RoboDK station: kr30 cnc 070119 curve 7 axis test 2.rdk

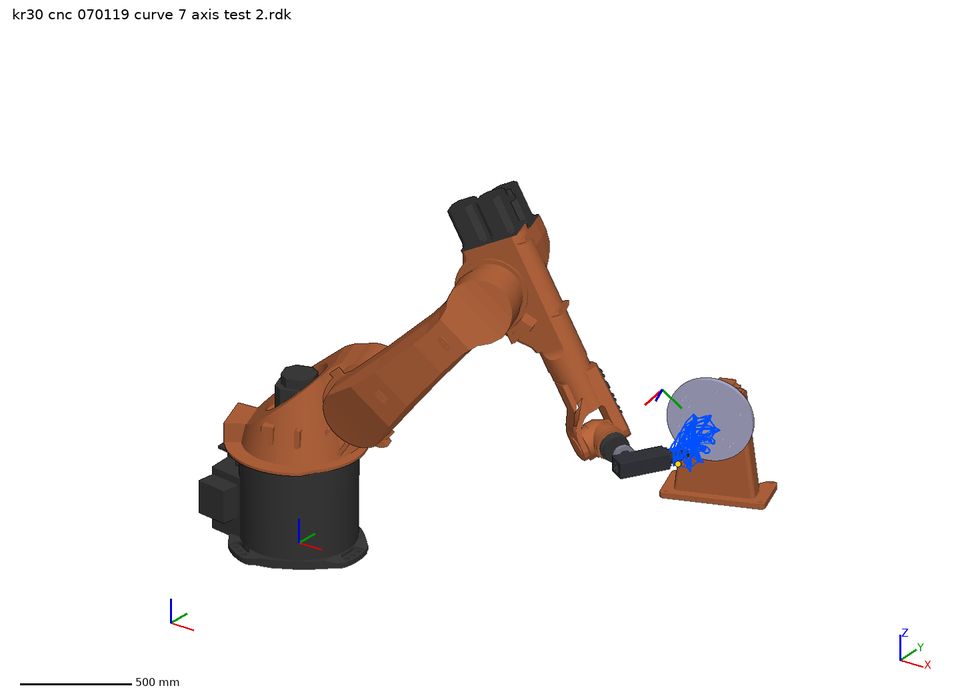
[picture v0: the station drawn from its stored meshes, robots at their saved joint values, targets as dots, program paths as lines]
Station kr30 cnc 070119 curve 7 axis test 2. Poses are relative to the parent item; angles as X-Y-Z fixed-axis rotations.
  - machining project Curve settings: C:/Temp/temp3/RhinoProject.stl | rotZ(0) | rotX(0)*rotY(0) | rotz(0) | onStart | onPathStart | onApproach | onPoint | onRetract | onFinish | onPathFinish | M_RunCode(%1)
  - frame KUKA KP1 MD250 Base at (0, 1000, 0) mm
    - robot KUKA KP1 MD250: 1 axes, payload 250 kg
        modified DH rows (alpha deg, a mm, theta deg, d mm): 0, 0, 0, 0
        base shift (1750, 1710, 820) mm, rotated rx 0 ry 90 rz -70 deg
        joint limits [-3600] to [3600]; home [0]; saved at [-1842.679]
      - frame Reference Rhino at (0, -260, 100) mm
        - object RhinoPart at (0, 0, 0) mm
  - frame KUKA KR 30 HA Base at (0, 2000, 0) mm
    - robot KUKA KR 30 HA: 6 axes, payload 30 kg, reach 2033 mm, repeatability 0.05 mm, weight 665 kg
        modified DH rows (alpha deg, a mm, theta deg, d mm): 0, 0, 0, 815; -90, 350, 0, 0; 0, 850, -90, 0; -90, 145, 0, 820; 90, 0, 0, 0; -90, 0, 180, 170
        joint limits [-185, -135, -120, -350, -119, -350] to [185, 35, 158, 350, 119, 350]; home [0, -90, 90, 0, 0, 0]; saved at [-17.768, -46.202, 111.125, 129.427, 73.448, 109.11]
      - tool 1/2" End Mill TCP, TCP at (337.71, -2.2, 160.57) mm, rotated rx 0 ry 90 rz 0 deg, size 415.8 x 102 x 153.6 mm
  - machining project RhinoPart Settings: rotZ(0) | rotX(0)*rotY(50) | rotz(0) | onStart | onPathStart | onApproach | onPoint | onRetract | onFinish | onPathFinish | M_RunCode(%1)
  - program RhinoPart (1340 instructions, listed below)
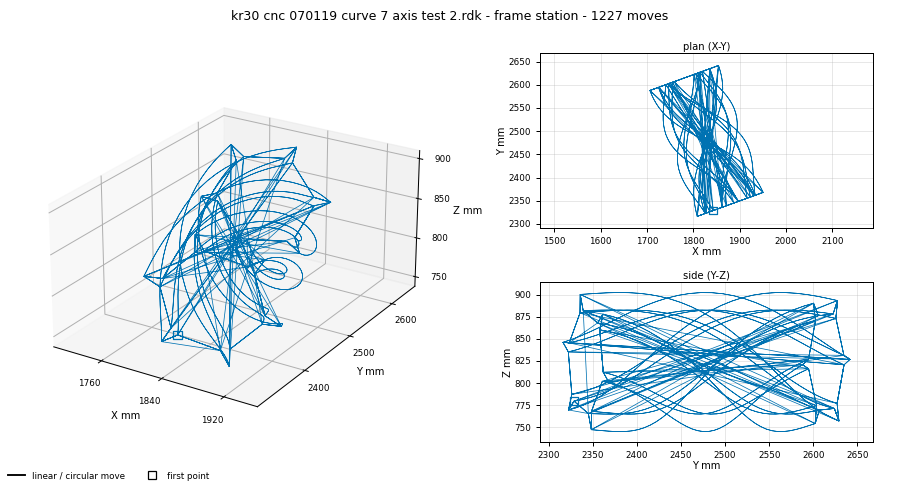
[picture p0: tool path of kr30 cnc 070119 curve 7 axis test 2.rdk in frame station, 1227 of 1227 moves have a stored position in this frame; points joined in program order, loops and branches not executed]

--- program RhinoPart (robot KUKA KR 30 HA) ---
  Set Ref.: Reference Rhino
  Set Tool: 1/2" End Mill TCP
  Show 1/2" End Mill TCP
  Set speed (1000.0 mm/s)
  MoveJ 1 to (58.93, 255.88, 290) mm, rotated rx 180 ry 50 rz -94 deg; joints [-8.613, -45.973, 108.773, 138.077, 69.074, 107.782, 4.002]
  MoveL 2 to (58.93, 255.88, 290) mm, rotated rx 180 ry 50 rz -94 deg; joints [-8.613, -45.973, 108.773, 138.077, 69.074, 107.782, 4.002]
  MoveL 3 to (58.93, 255.88, 290) mm, rotated rx 180 ry 50 rz -94 deg; joints [-8.613, -45.973, 108.773, 138.077, 69.074, 107.782, 4.002]
  Set speed (60.0 mm/s)
  MoveL 4 to (37.11, 300.24, 290) mm, rotated rx 180 ry 50 rz -42.69 deg; joints [-8.613, -46.208, 108.79, 138.021, 68.912, 107.938, -47.315]
  MoveL 5 to (-37.11, 208.63, 290) mm, rotated rx 180 ry 50 rz 144.16 deg; joints [-8.613, -45.739, 108.754, 138.132, 69.233, 107.629, 125.844]
  Set speed (60.0 mm/s)
  MoveL 6 to (-58.93, 252.99, 290) mm, rotated rx 180 ry 50 rz 96.78 deg; joints [-8.613, -45.958, 108.772, 138.081, 69.084, 107.773, 173.216]
  MoveL 7 to (21.11, 199.39, 290) mm, rotated rx 180 ry 50 rz -160.79 deg; joints [-8.613, -45.696, 108.75, 138.142, 69.263, 107.6, 70.794]
  Set speed (60.0 mm/s)
  MoveL 8 to (34.79, 183.72, 290) mm, rotated rx -180 ry 50 rz -155.49 deg; joints [-8.613, -44.618, 108.643, 138.382, 69.987, 106.912, 65.485]
  MoveL 9 to (21.11, 199.39, 290) mm, rotated rx -180 ry 50 rz -160.79 deg; joints [-8.613, -45.696, 108.75, 138.142, 69.263, 107.6, 70.794]
  Set speed (60.0 mm/s)
  MoveL 10 to (-28.22, 202.67, 290) mm, rotated rx 180 ry 50 rz 153.79 deg; joints [-8.613, -45.711, 108.751, 138.138, 69.253, 107.611, 116.207]
  MoveL 11 to (-43.85, 188.95, 290) mm, rotated rx -180 ry 50 rz 148.32 deg; joints [-8.613, -44.637, 108.645, 138.378, 69.974, 106.924, 121.679]
  Set speed (60.0 mm/s)
  MoveL 12 to (-28.22, 202.67, 290) mm, rotated rx -180 ry 50 rz 153.79 deg; joints [-8.613, -45.711, 108.751, 138.138, 69.253, 107.611, 116.207]
  MoveL 13 to (-43.85, 188.95, 290) mm, rotated rx -180 ry 50 rz 148.32 deg; joints [-8.613, -44.637, 108.645, 138.378, 69.974, 106.924, 121.679]
  Set speed (60.0 mm/s)
  MoveL 14 to (-37.11, 208.63, 290) mm, rotated rx 180 ry 50 rz 144.16 deg; joints [-8.613, -45.739, 108.754, 138.132, 69.233, 107.629, 125.844]
  MoveL 15 to (-78.63, 259.66, 290) mm, rotated rx -180 ry 50 rz 90.25 deg; joints [-8.613, -44.905, 108.674, 138.32, 69.797, 107.092, 179.755]
  Set speed (60.0 mm/s)
  MoveL 16 to (-58.93, 252.99, 290) mm, rotated rx 180 ry 50 rz 96.78 deg; joints [-8.613, -45.958, 108.772, 138.081, 69.084, 107.773, 173.216]
  MoveL 17 to (-78.63, 259.66, 290) mm, rotated rx 180 ry 50 rz 90.25 deg; joints [-8.613, -44.905, 108.674, 138.32, 69.797, 107.092, 179.755]
  Set speed (60.0 mm/s)
  MoveL 18 to (-58.22, 263.67, 290) mm, rotated rx -180 ry 50 rz 86.39 deg; joints [-8.613, -46.013, 108.776, 138.068, 69.046, 107.809, 183.606]
  MoveL 19 to (-30.72, 304.75, 290) mm, rotated rx -180 ry 50 rz 34.47 deg; joints [-8.613, -46.233, 108.792, 138.015, 68.894, 107.955, 235.533]
  Set speed (60.0 mm/s)
  MoveL 20 to (-58.22, 263.67, 290) mm, rotated rx -180 ry 50 rz 86.39 deg; joints [-8.613, -46.013, 108.776, 138.068, 69.046, 107.809, 183.606]
  MoveL 21 to (-30.72, 304.75, 290) mm, rotated rx -180 ry 50 rz 34.47 deg; joints [-8.613, -46.233, 108.792, 138.015, 68.894, 107.955, 235.533]
  Set speed (60.0 mm/s)
  MoveL 22 to (-34.79, 325.15, 290) mm, rotated rx 180 ry 50 rz 28.1 deg; joints [-8.613, -45.167, 108.701, 138.262, 69.621, 107.259, 241.899]
  MoveL 23 to (-21.11, 309.47, 290) mm, rotated rx 180 ry 50 rz 23.11 deg; joints [-8.613, -46.26, 108.794, 138.009, 68.876, 107.972, 246.89]
  Set speed (60.0 mm/s)
  MoveL 24 to (-34.79, 325.15, 290) mm, rotated rx 180 ry 50 rz 28.1 deg; joints [-8.613, -45.167, 108.701, 138.262, 69.621, 107.259, 241.899]
  MoveL 25 to (-21.11, 309.47, 290) mm, rotated rx 180 ry 50 rz 23.11 deg; joints [-8.613, -46.26, 108.794, 138.009, 68.876, 107.972, 246.89]
  Set speed (60.0 mm/s)
  MoveL 26 to (28.22, 306.19, 290) mm, rotated rx 180 ry 50 rz -31.42 deg; joints [-8.613, -46.241, 108.793, 138.013, 68.889, 107.96, 301.418]
  MoveL 27 to (43.85, 319.91, 290) mm, rotated rx 180 ry 50 rz -36.2 deg; joints [-8.613, -45.145, 108.699, 138.267, 69.635, 107.245, 306.197]
  Set speed (60.0 mm/s)
  MoveL 28 to (28.22, 306.19, 290) mm, rotated rx 180 ry 50 rz -31.42 deg; joints [-8.613, -46.241, 108.793, 138.013, 68.889, 107.96, 301.418]
  MoveL 29 to (43.85, 319.91, 290) mm, rotated rx 180 ry 50 rz -36.2 deg; joints [-8.613, -45.145, 108.699, 138.267, 69.635, 107.245, 306.197]
  Set speed (60.0 mm/s)
  MoveL 30 to (37.11, 300.24, 290) mm, rotated rx -180 ry 50 rz -42.69 deg; joints [-8.613, -46.208, 108.79, 138.021, 68.912, 107.938, 312.685]
  MoveL 31 to (78.63, 249.2, 290) mm, rotated rx -180 ry 50 rz -97.82 deg; joints [-8.613, -44.864, 108.67, 138.329, 69.824, 107.066, 367.819]
  Set speed (60.0 mm/s)
  MoveL 32 to (58.93, 255.88, 290) mm, rotated rx 180 ry 50 rz -94 deg; joints [-8.613, -45.973, 108.773, 138.077, 69.074, 107.782, 364.002]
  MoveL 33 to (78.63, 249.2, 290) mm, rotated rx 180 ry 50 rz -97.82 deg; joints [-8.613, -44.864, 108.67, 138.329, 69.824, 107.066, 367.819]
  Set speed (60.0 mm/s)
  MoveL 34 to (58.22, 245.2, 290) mm, rotated rx -180 ry 50 rz -104.27 deg; joints [-8.613, -45.919, 108.769, 138.09, 69.111, 107.747, 374.265]
  MoveL 35 to (30.72, 204.12, 290) mm, rotated rx -180 ry 50 rz -151.2 deg; joints [-8.613, -45.718, 108.752, 138.137, 69.248, 107.615, 421.204]
  Set speed (60.0 mm/s)
  MoveL 36 to (58.22, 245.2, 290) mm, rotated rx -180 ry 50 rz -104.27 deg; joints [-8.613, -45.919, 108.769, 138.09, 69.111, 107.747, 374.265]
  MoveL 37 to (30.72, 204.12, 290) mm, rotated rx -180 ry 50 rz -151.2 deg; joints [-8.613, -45.718, 108.752, 138.137, 69.248, 107.615, 421.204]
  Set speed (60.0 mm/s)
  MoveL 38 to (34.79, 183.72, 290) mm, rotated rx 180 ry 50 rz -155.49 deg; joints [-8.613, -44.618, 108.643, 138.382, 69.987, 106.912, 425.485]
  MoveL 39 to (-37.62, 299.82, 0) mm, rotated rx 180 ry 50 rz 43.38 deg; joints [-20.194, -47.371, 111.315, 126.82, 73.668, 110.587, 586.623]
  Set speed (60.0 mm/s)
  MoveL 40 to (10.16, 312.5, 0) mm, rotated rx 180 ry 50 rz -10.95 deg; joints [-20.194, -47.443, 111.32, 126.804, 73.628, 110.643, 640.953]
  MoveL 41 to (-37.62, 299.82, 0) mm, rotated rx 180 ry 50 rz 43.38 deg; joints [-20.194, -47.371, 111.315, 126.82, 73.668, 110.587, 586.623]
  Set speed (60.0 mm/s)
  MoveL 42 to (-55.59, 310.29, 0) mm, rotated rx 180 ry 50 rz 47.87 deg; joints [-20.194, -46.242, 111.219, 127.057, 74.288, 109.729, 582.13]
  MoveL 43 to (-45.21, 292.27, 0) mm, rotated rx -180 ry 50 rz 54.48 deg; joints [-20.194, -47.328, 111.312, 126.829, 73.692, 110.554, 575.516]
  Set speed (60.0 mm/s)
  MoveL 44 to (-55.59, 310.29, 0) mm, rotated rx 180 ry 50 rz 47.87 deg; joints [-20.194, -46.242, 111.219, 127.057, 74.288, 109.729, 582.13]
  MoveL 45 to (-45.21, 292.27, 0) mm, rotated rx -180 ry 50 rz 54.48 deg; joints [-20.194, -47.328, 111.312, 126.829, 73.692, 110.554, 575.516]
  Set speed (60.0 mm/s)
  MoveL 46 to (-58.12, 244.54, 0) mm, rotated rx -180 ry 50 rz 104.89 deg; joints [-20.194, -47.073, 111.293, 126.884, 73.834, 110.357, 525.106]
  MoveL 47 to (-76.17, 234.21, 0) mm, rotated rx 180 ry 50 rz 108.7 deg; joints [-20.194, -45.935, 111.187, 127.118, 74.455, 109.5, 521.297]
  Set speed (60.0 mm/s)
  MoveL 48 to (-58.12, 244.54, 0) mm, rotated rx 180 ry 50 rz 104.89 deg; joints [-20.194, -47.073, 111.293, 126.884, 73.834, 110.357, 525.106]
  MoveL 49 to (-76.17, 234.21, 0) mm, rotated rx 180 ry 50 rz 108.7 deg; joints [-20.194, -45.935, 111.187, 127.118, 74.455, 109.5, 521.297]
  Set speed (60.0 mm/s)
  MoveL 50 to (-55.37, 234.2, 0) mm, rotated rx 180 ry 50 rz 114.99 deg; joints [-20.194, -47.02, 111.288, 126.896, 73.863, 110.316, 515.014]
  MoveL 51 to (-20.49, 199.16, 0) mm, rotated rx -180 ry 50 rz 161.39 deg; joints [-20.194, -46.846, 111.274, 126.932, 73.959, 110.184, 468.615]
  Set speed (60.0 mm/s)
  MoveL 52 to (-55.37, 234.2, 0) mm, rotated rx 180 ry 50 rz 114.99 deg; joints [-20.194, -47.02, 111.288, 126.896, 73.863, 110.316, 515.014]
  MoveL 53 to (-20.49, 199.16, 0) mm, rotated rx -180 ry 50 rz 161.39 deg; joints [-20.194, -46.846, 111.274, 126.932, 73.959, 110.184, 468.615]
  Set speed (60.0 mm/s)
  MoveL 54 to (-20.57, 178.36, 0) mm, rotated rx -180 ry 50 rz 165.86 deg; joints [-20.194, -45.722, 111.164, 127.16, 74.569, 109.343, 464.144]
  MoveL 55 to (-10.16, 196.36, 0) mm, rotated rx -180 ry 50 rz 170.93 deg; joints [-20.194, -46.832, 111.273, 126.935, 73.966, 110.173, 459.071]
  Set speed (60.0 mm/s)
  MoveL 56 to (-20.57, 178.36, 0) mm, rotated rx -180 ry 50 rz 165.86 deg; joints [-20.194, -45.722, 111.164, 127.16, 74.569, 109.343, 464.144]
  MoveL 57 to (-10.16, 196.36, 0) mm, rotated rx -180 ry 50 rz 170.93 deg; joints [-20.194, -46.832, 111.273, 126.935, 73.966, 110.173, 459.071]
  Set speed (60.0 mm/s)
  MoveL 58 to (37.62, 209.05, 0) mm, rotated rx 180 ry 50 rz -143.56 deg; joints [-20.194, -46.894, 111.278, 126.922, 73.932, 110.22, 413.558]
  MoveL 59 to (55.59, 198.58, 0) mm, rotated rx 180 ry 50 rz -137.85 deg; joints [-20.194, -45.798, 111.172, 127.145, 74.528, 109.399, 407.85]
  Set speed (60.0 mm/s)
  MoveL 60 to (37.62, 209.05, 0) mm, rotated rx 180 ry 50 rz -143.56 deg; joints [-20.194, -46.894, 111.278, 126.922, 73.932, 110.22, 413.558]
  MoveL 61 to (55.59, 198.58, 0) mm, rotated rx 180 ry 50 rz -137.85 deg; joints [-20.194, -45.798, 111.172, 127.145, 74.528, 109.399, 407.85]
  Set speed (60.0 mm/s)
  MoveL 62 to (45.21, 216.6, 0) mm, rotated rx -180 ry 50 rz -133.83 deg; joints [-20.194, -46.931, 111.281, 126.914, 73.912, 110.249, 403.831]
  MoveL 63 to (58.12, 264.32, 0) mm, rotated rx -180 ry 50 rz -85.75 deg; joints [-20.194, -47.176, 111.301, 126.862, 73.776, 110.437, 355.746]
  Set speed (60.0 mm/s)
  MoveL 64 to (45.21, 216.6, 0) mm, rotated rx 180 ry 50 rz -133.83 deg; joints [-20.194, -46.931, 111.281, 126.914, 73.912, 110.249, 403.831]
  MoveL 65 to (58.12, 264.32, 0) mm, rotated rx -180 ry 50 rz -85.75 deg; joints [-20.194, -47.176, 111.301, 126.862, 73.776, 110.437, 355.746]
  Set speed (60.0 mm/s)
  MoveL 66 to (76.17, 274.65, 0) mm, rotated rx 180 ry 50 rz -79.11 deg; joints [-20.194, -46.096, 111.204, 127.086, 74.368, 109.619, 349.111]
  MoveL 67 to (55.37, 274.67, 0) mm, rotated rx 180 ry 50 rz -75.16 deg; joints [-20.194, -47.232, 111.305, 126.85, 73.745, 110.479, 345.162]
  Set speed (60.0 mm/s)
  MoveL 68 to (76.17, 274.65, 0) mm, rotated rx 180 ry 50 rz -79.11 deg; joints [-20.194, -46.096, 111.204, 127.086, 74.368, 109.619, 349.111]
  MoveL 69 to (55.37, 274.67, 0) mm, rotated rx 180 ry 50 rz -75.16 deg; joints [-20.194, -47.232, 111.305, 126.85, 73.745, 110.479, 345.162]
  Set speed (60.0 mm/s)
  MoveL 70 to (20.49, 309.71, 0) mm, rotated rx -180 ry 50 rz -22.4 deg; joints [-20.194, -47.427, 111.319, 126.808, 73.637, 110.631, 292.405]
  MoveL 71 to (20.57, 330.51, 0) mm, rotated rx -180 ry 50 rz -16.27 deg; joints [-20.194, -46.328, 111.227, 127.04, 74.242, 109.792, 286.267]
  Set speed (60.0 mm/s)
  MoveL 72 to (20.49, 309.71, 0) mm, rotated rx -180 ry 50 rz -22.4 deg; joints [-20.194, -47.427, 111.319, 126.808, 73.637, 110.631, 292.405]
  MoveL 73 to (20.57, 330.51, 0) mm, rotated rx -180 ry 50 rz -16.27 deg; joints [-20.194, -46.328, 111.227, 127.04, 74.242, 109.792, 286.267]
  Set speed (60.0 mm/s)
  MoveL 74 to (10.16, 312.5, 0) mm, rotated rx 180 ry 50 rz -10.95 deg; joints [-20.194, -47.443, 111.32, 126.804, 73.628, 110.643, 280.953]
  MoveL 75 to (-37.62, 299.82, 0) mm, rotated rx 180 ry 50 rz 43.38 deg; joints [-20.194, -47.371, 111.315, 126.82, 73.668, 110.587, 226.623]
  Set speed (60.0 mm/s)
  MoveL 76 to (-40.85, 296.93, 10) mm, rotated rx 180 ry 50 rz 47.89 deg; joints [-19.79, -47.354, 111.314, 127.219, 73.535, 110.463, 222.114]
  MoveL 77 to (-44.15, 293.5, 20) mm, rotated rx -180 ry 50 rz 52.81 deg; joints [-19.385, -47.332, 111.306, 127.618, 73.403, 110.338, 217.19]
  MoveL 78 to (-47.39, 289.5, 30) mm, rotated rx -180 ry 50 rz 58.1 deg; joints [-18.981, -47.304, 111.292, 128.017, 73.271, 110.213, 211.9]
  MoveL 79 to (-50.45, 284.92, 40) mm, rotated rx 180 ry 50 rz 63.71 deg; joints [-18.576, -47.27, 111.271, 128.417, 73.14, 110.088, 206.29]
  MoveL 80 to (-53.21, 279.8, 50) mm, rotated rx 180 ry 50 rz 69.59 deg; joints [-18.172, -47.231, 111.244, 128.817, 73.01, 109.962, 200.409]
  MoveL 81 to (-55.55, 274.16, 60) mm, rotated rx -180 ry 50 rz 75.7 deg; joints [-17.768, -47.186, 111.211, 129.217, 72.879, 109.836, 194.303]
  MoveL 82 to (-57.35, 268.08, 70) mm, rotated rx 180 ry 50 rz 81.99 deg; joints [-17.364, -47.136, 111.171, 129.617, 72.749, 109.711, 188.015]
  MoveL 83 to (-58.51, 261.62, 80) mm, rotated rx 180 ry 50 rz 88.41 deg; joints [-16.96, -47.082, 111.125, 130.017, 72.618, 109.586, 181.589]
  MoveL 84 to (-58.95, 254.91, 90) mm, rotated rx 180 ry 50 rz 94.94 deg; joints [-16.557, -47.024, 111.072, 130.417, 72.487, 109.462, 175.064]
  MoveL 85 to (-58.6, 248.05, 100) mm, rotated rx 180 ry 50 rz 101.52 deg; joints [-16.154, -46.962, 111.013, 130.816, 72.355, 109.339, 168.479]
  MoveL 86 to (-57.44, 241.19, 110) mm, rotated rx 180 ry 50 rz 108.13 deg; joints [-15.751, -46.899, 110.948, 131.215, 72.221, 109.219, 161.868]
  MoveL 87 to (-55.46, 234.45, 120) mm, rotated rx 180 ry 50 rz 114.74 deg; joints [-15.349, -46.833, 110.877, 131.613, 72.086, 109.101, 155.264]
  MoveL 88 to (-52.68, 227.97, 130) mm, rotated rx 180 ry 50 rz 121.3 deg; joints [-14.948, -46.766, 110.8, 132.009, 71.948, 108.986, 148.698]
  MoveL 89 to (-49.15, 221.88, 140) mm, rotated rx 180 ry 50 rz 127.8 deg; joints [-14.546, -46.699, 110.716, 132.405, 71.807, 108.874, 142.199]
  MoveL 90 to (-44.94, 216.28, 150) mm, rotated rx -180 ry 50 rz 134.21 deg; joints [-14.146, -46.632, 110.627, 132.799, 71.663, 108.766, 135.793]
  MoveL 91 to (-40.17, 211.29, 160) mm, rotated rx 180 ry 50 rz 140.49 deg; joints [-13.746, -46.565, 110.532, 133.191, 71.515, 108.662, 129.508]
  MoveL 92 to (-34.94, 206.95, 170) mm, rotated rx 180 ry 50 rz 146.63 deg; joints [-13.346, -46.498, 110.431, 133.582, 71.364, 108.561, 123.368]
  MoveL 93 to (-29.38, 203.32, 180) mm, rotated rx 180 ry 50 rz 152.6 deg; joints [-12.947, -46.432, 110.323, 133.971, 71.208, 108.465, 117.399]
  MoveL 94 to (-23.62, 200.42, 190) mm, rotated rx 180 ry 50 rz 158.37 deg; joints [-12.549, -46.367, 110.21, 134.359, 71.049, 108.372, 111.627]
  MoveL 95 to (-17.8, 198.23, 200) mm, rotated rx -180 ry 50 rz 163.92 deg; joints [-12.152, -46.303, 110.091, 134.744, 70.886, 108.283, 106.077]
  MoveL 96 to (-12.04, 196.73, 210) mm, rotated rx 180 ry 50 rz 169.22 deg; joints [-11.755, -46.239, 109.966, 135.128, 70.718, 108.198, 100.776]
  MoveL 97 to (-6.46, 195.84, 220) mm, rotated rx 180 ry 50 rz 174.25 deg; joints [-11.359, -46.175, 109.836, 135.51, 70.547, 108.115, 95.751]
  MoveL 98 to (-1.16, 195.49, 230) mm, rotated rx -180 ry 50 rz 178.97 deg; joints [-10.964, -46.111, 109.699, 135.891, 70.373, 108.036, 91.029]
  MoveL 99 to (3.78, 195.6, 240) mm, rotated rx -180 ry 50 rz -176.64 deg; joints [-10.57, -46.047, 109.556, 136.27, 70.195, 107.959, 86.641]
  MoveL 100 to (8.28, 196.07, 250) mm, rotated rx -180 ry 50 rz -172.62 deg; joints [-10.177, -45.981, 109.407, 136.647, 70.013, 107.885, 82.617]
  MoveL 101 to (12.3, 196.78, 260) mm, rotated rx 180 ry 50 rz -168.99 deg; joints [-9.784, -45.913, 109.252, 137.023, 69.829, 107.812, 78.987]
  MoveL 102 to (15.8, 197.64, 270) mm, rotated rx 180 ry 50 rz -165.79 deg; joints [-9.393, -45.843, 109.091, 137.397, 69.643, 107.74, 75.785]
  MoveL 103 to (18.74, 198.54, 280) mm, rotated rx 180 ry 50 rz -163.04 deg; joints [-9.003, -45.771, 108.924, 137.77, 69.454, 107.67, 73.043]
  MoveL 104 to (21.11, 199.39, 290) mm, rotated rx 180 ry 50 rz -160.79 deg; joints [-8.613, -45.696, 108.75, 138.142, 69.263, 107.6, 70.794]
  MoveL 105 to (10.16, 312.5, 0) mm, rotated rx 180 ry 50 rz -10.95 deg; joints [-20.194, -47.443, 111.32, 126.804, 73.628, 110.643, -79.047]
  Set speed (60.0 mm/s)
  MoveL 106 to (-37.62, 299.82, 0) mm, rotated rx 180 ry 50 rz 43.38 deg; joints [-20.194, -47.371, 111.315, 126.82, 73.668, 110.587, -133.377]
  MoveL 107 to (-28.22, 202.67, 290) mm, rotated rx -180 ry 50 rz 153.79 deg; joints [-8.613, -45.711, 108.751, 138.138, 69.253, 107.611, -243.793]
  Set speed (60.0 mm/s)
  MoveL 108 to (21.11, 199.39, 290) mm, rotated rx -180 ry 50 rz -160.79 deg; joints [-8.613, -45.696, 108.75, 138.142, 69.263, 107.6, -289.206]
  MoveL 109 to (-28.22, 202.67, 290) mm, rotated rx 180 ry 50 rz 153.79 deg; joints [-8.613, -45.711, 108.751, 138.138, 69.253, 107.611, -243.793]
  Set speed (60.0 mm/s)
  MoveL 110 to (-30.4, 203.93, 280) mm, rotated rx 180 ry 50 rz 151.53 deg; joints [-9.003, -45.797, 108.926, 137.764, 69.437, 107.687, -241.533]
  MoveL 111 to (-33, 205.58, 270) mm, rotated rx 180 ry 50 rz 148.77 deg; joints [-9.393, -45.881, 109.094, 137.388, 69.617, 107.765, -238.768]
  MoveL 112 to (-35.92, 207.69, 260) mm, rotated rx -180 ry 50 rz 145.53 deg; joints [-9.784, -45.965, 109.256, 137.011, 69.795, 107.846, -235.528]
  MoveL 113 to (-39.07, 210.28, 250) mm, rotated rx 180 ry 50 rz 141.84 deg; joints [-10.177, -46.049, 109.413, 136.631, 69.968, 107.93, -231.841]
  MoveL 114 to (-42.34, 213.41, 240) mm, rotated rx 180 ry 50 rz 137.73 deg; joints [-10.57, -46.132, 109.563, 136.25, 70.138, 108.017, -227.735]
  MoveL 115 to (-45.62, 217.1, 230) mm, rotated rx -180 ry 50 rz 133.24 deg; joints [-10.964, -46.215, 109.708, 135.867, 70.304, 108.106, -223.236]
  MoveL 116 to (-48.8, 221.36, 220) mm, rotated rx 180 ry 50 rz 128.37 deg; joints [-11.359, -46.299, 109.846, 135.482, 70.467, 108.199, -218.371]
  MoveL 117 to (-51.74, 226.19, 210) mm, rotated rx 180 ry 50 rz 123.16 deg; joints [-11.755, -46.382, 109.978, 135.096, 70.625, 108.296, -213.164]
  MoveL 118 to (-54.33, 231.55, 200) mm, rotated rx 180 ry 50 rz 117.64 deg; joints [-12.152, -46.466, 110.105, 134.707, 70.781, 108.395, -207.64]
  MoveL 119 to (-56.44, 237.4, 190) mm, rotated rx 180 ry 50 rz 111.82 deg; joints [-12.549, -46.549, 110.225, 134.318, 70.932, 108.498, -201.825]
  MoveL 120 to (-57.96, 243.66, 180) mm, rotated rx -180 ry 50 rz 105.74 deg; joints [-12.947, -46.632, 110.34, 133.926, 71.081, 108.604, -195.742]
  MoveL 121 to (-58.8, 250.25, 170) mm, rotated rx -180 ry 50 rz 99.42 deg; joints [-13.346, -46.715, 110.448, 133.533, 71.226, 108.713, -189.418]
  MoveL 122 to (-58.89, 257.04, 160) mm, rotated rx 180 ry 50 rz 92.88 deg; joints [-13.746, -46.795, 110.55, 133.139, 71.37, 108.825, -182.877]
  MoveL 123 to (-58.18, 263.92, 150) mm, rotated rx 180 ry 50 rz 86.15 deg; joints [-14.146, -46.874, 110.646, 132.744, 71.511, 108.939, -176.149]
  MoveL 124 to (-56.65, 270.74, 140) mm, rotated rx 180 ry 50 rz 79.26 deg; joints [-14.546, -46.951, 110.736, 132.348, 71.65, 109.055, -169.263]
  MoveL 125 to (-54.3, 277.38, 130) mm, rotated rx 180 ry 50 rz 72.25 deg; joints [-14.948, -47.023, 110.82, 131.951, 71.789, 109.171, -162.251]
  MoveL 126 to (-51.17, 283.7, 120) mm, rotated rx 180 ry 50 rz 65.15 deg; joints [-15.349, -47.092, 110.897, 131.554, 71.927, 109.289, -155.149]
  MoveL 127 to (-47.33, 289.58, 110) mm, rotated rx -180 ry 50 rz 57.99 deg; joints [-15.751, -47.156, 110.968, 131.157, 72.065, 109.407, -147.994]
  MoveL 128 to (-42.85, 294.92, 100) mm, rotated rx 180 ry 50 rz 50.83 deg; joints [-16.154, -47.214, 111.032, 130.76, 72.203, 109.524, -140.828]
  MoveL 129 to (-37.86, 299.62, 90) mm, rotated rx -180 ry 50 rz 43.7 deg; joints [-16.557, -47.266, 111.09, 130.363, 72.342, 109.641, -133.695]
  MoveL 130 to (-32.46, 303.64, 80) mm, rotated rx -180 ry 50 rz 36.64 deg; joints [-16.96, -47.312, 111.141, 129.966, 72.482, 109.757, -126.643]
  MoveL 131 to (-26.8, 306.94, 70) mm, rotated rx -180 ry 50 rz 29.72 deg; joints [-17.364, -47.351, 111.186, 129.569, 72.622, 109.871, -119.72]
  MoveL 132 to (-21, 309.52, 60) mm, rotated rx 180 ry 50 rz 22.98 deg; joints [-17.768, -47.383, 111.225, 129.173, 72.764, 109.984, -112.977]
  MoveL 133 to (-15.19, 311.39, 50) mm, rotated rx -180 ry 50 rz 16.46 deg; joints [-18.172, -47.408, 111.257, 128.777, 72.907, 110.096, -106.464]
  MoveL 134 to (-9.5, 312.61, 40) mm, rotated rx 180 ry 50 rz 10.23 deg; joints [-18.576, -47.426, 111.282, 128.382, 73.05, 110.207, -100.231]
  MoveL 135 to (-4.03, 313.25, 30) mm, rotated rx -180 ry 50 rz 4.33 deg; joints [-18.981, -47.439, 111.301, 127.987, 73.194, 110.316, -94.327]
  MoveL 136 to (1.12, 313.37, 20) mm, rotated rx 180 ry 50 rz -1.2 deg; joints [-19.385, -47.445, 111.314, 127.593, 73.339, 110.425, -88.799]
  MoveL 137 to (5.87, 313.09, 10) mm, rotated rx -180 ry 50 rz -6.31 deg; joints [-19.79, -47.446, 111.32, 127.198, 73.484, 110.534, -83.692]
  MoveL 138 to (10.16, 312.5, 0) mm, rotated rx 180 ry 50 rz -10.95 deg; joints [-20.194, -47.443, 111.32, 126.804, 73.628, 110.643, -79.047]
  MoveL 139 to (-37.62, 299.82, 0) mm, rotated rx 180 ry 50 rz 43.38 deg; joints [-20.194, -47.371, 111.315, 126.82, 73.668, 110.587, -133.377]
  Set speed (60.0 mm/s)
  MoveL 140 to (-40.85, 296.93, 10) mm, rotated rx 180 ry 50 rz 47.89 deg; joints [-19.79, -47.354, 111.314, 127.219, 73.535, 110.463, -137.886]
  MoveL 141 to (-44.15, 293.5, 20) mm, rotated rx -180 ry 50 rz 52.81 deg; joints [-19.385, -47.332, 111.306, 127.618, 73.403, 110.338, -142.81]
  MoveL 142 to (-47.39, 289.5, 30) mm, rotated rx -180 ry 50 rz 58.1 deg; joints [-18.981, -47.304, 111.292, 128.017, 73.271, 110.213, -148.1]
  MoveL 143 to (-50.45, 284.92, 40) mm, rotated rx 180 ry 50 rz 63.71 deg; joints [-18.576, -47.27, 111.271, 128.417, 73.14, 110.088, -153.71]
  MoveL 144 to (-53.21, 279.8, 50) mm, rotated rx 180 ry 50 rz 69.59 deg; joints [-18.172, -47.231, 111.244, 128.817, 73.01, 109.962, -159.591]
  MoveL 145 to (-55.55, 274.16, 60) mm, rotated rx -180 ry 50 rz 75.7 deg; joints [-17.768, -47.186, 111.211, 129.217, 72.879, 109.836, -165.697]
  MoveL 146 to (-57.35, 268.08, 70) mm, rotated rx 180 ry 50 rz 81.99 deg; joints [-17.364, -47.136, 111.171, 129.617, 72.749, 109.711, -171.985]
  MoveL 147 to (-58.51, 261.62, 80) mm, rotated rx -180 ry 50 rz 88.41 deg; joints [-16.96, -47.082, 111.125, 130.017, 72.618, 109.586, -178.411]
  MoveL 148 to (-58.95, 254.91, 90) mm, rotated rx 180 ry 50 rz 94.94 deg; joints [-16.557, -47.024, 111.072, 130.417, 72.487, 109.462, -184.936]
  MoveL 149 to (-58.6, 248.05, 100) mm, rotated rx 180 ry 50 rz 101.52 deg; joints [-16.154, -46.962, 111.013, 130.816, 72.355, 109.339, -191.521]
  MoveL 150 to (-57.44, 241.19, 110) mm, rotated rx 180 ry 50 rz 108.13 deg; joints [-15.751, -46.899, 110.948, 131.215, 72.221, 109.219, -198.132]
  MoveL 151 to (-55.46, 234.45, 120) mm, rotated rx 180 ry 50 rz 114.74 deg; joints [-15.349, -46.833, 110.877, 131.613, 72.086, 109.101, -204.736]
  MoveL 152 to (-52.68, 227.97, 130) mm, rotated rx 180 ry 50 rz 121.3 deg; joints [-14.948, -46.766, 110.8, 132.009, 71.948, 108.986, -211.302]
  MoveL 153 to (-49.15, 221.88, 140) mm, rotated rx 180 ry 50 rz 127.8 deg; joints [-14.546, -46.699, 110.716, 132.405, 71.807, 108.874, -217.801]
  MoveL 154 to (-44.94, 216.28, 150) mm, rotated rx 180 ry 50 rz 134.21 deg; joints [-14.146, -46.632, 110.627, 132.799, 71.663, 108.766, -224.207]
  MoveL 155 to (-40.17, 211.29, 160) mm, rotated rx 180 ry 50 rz 140.49 deg; joints [-13.746, -46.565, 110.532, 133.191, 71.515, 108.662, -230.492]
  MoveL 156 to (-34.94, 206.95, 170) mm, rotated rx 180 ry 50 rz 146.63 deg; joints [-13.346, -46.498, 110.431, 133.582, 71.364, 108.561, -236.632]
  MoveL 157 to (-29.38, 203.32, 180) mm, rotated rx 180 ry 50 rz 152.6 deg; joints [-12.947, -46.432, 110.323, 133.971, 71.208, 108.465, -242.601]
  MoveL 158 to (-23.62, 200.42, 190) mm, rotated rx -180 ry 50 rz 158.37 deg; joints [-12.549, -46.367, 110.21, 134.359, 71.049, 108.372, -248.373]
  MoveL 159 to (-17.8, 198.23, 200) mm, rotated rx -180 ry 50 rz 163.92 deg; joints [-12.152, -46.303, 110.091, 134.744, 70.886, 108.283, -253.923]
  MoveL 160 to (-12.04, 196.73, 210) mm, rotated rx 180 ry 50 rz 169.22 deg; joints [-11.755, -46.239, 109.966, 135.128, 70.718, 108.198, -259.224]
  MoveL 161 to (-6.46, 195.84, 220) mm, rotated rx -180 ry 50 rz 174.25 deg; joints [-11.359, -46.175, 109.836, 135.51, 70.547, 108.115, -264.249]
  MoveL 162 to (-1.16, 195.49, 230) mm, rotated rx 180 ry 50 rz 178.97 deg; joints [-10.964, -46.111, 109.699, 135.891, 70.373, 108.036, -268.971]
  MoveL 163 to (3.78, 195.6, 240) mm, rotated rx 180 ry 50 rz -176.64 deg; joints [-10.57, -46.047, 109.556, 136.27, 70.195, 107.959, -273.359]
  MoveL 164 to (8.28, 196.07, 250) mm, rotated rx 180 ry 50 rz -172.62 deg; joints [-10.177, -45.981, 109.407, 136.647, 70.013, 107.885, -277.383]
  MoveL 165 to (12.3, 196.78, 260) mm, rotated rx 180 ry 50 rz -168.99 deg; joints [-9.784, -45.913, 109.252, 137.023, 69.829, 107.812, -281.013]
  MoveL 166 to (15.8, 197.64, 270) mm, rotated rx 180 ry 50 rz -165.79 deg; joints [-9.393, -45.843, 109.091, 137.397, 69.643, 107.74, -284.215]
  MoveL 167 to (18.74, 198.54, 280) mm, rotated rx 180 ry 50 rz -163.04 deg; joints [-9.003, -45.771, 108.924, 137.77, 69.454, 107.67, -286.957]
  MoveL 168 to (21.11, 199.39, 290) mm, rotated rx 180 ry 50 rz -160.79 deg; joints [-8.613, -45.696, 108.75, 138.142, 69.263, 107.6, -289.206]
  MoveL 169 to (34.79, 183.72, 290) mm, rotated rx -180 ry 50 rz -155.49 deg; joints [-8.613, -44.618, 108.643, 138.382, 69.987, 106.912, -294.515]
  Set speed (60.0 mm/s)
  MoveL 170 to (21.11, 199.39, 290) mm, rotated rx -180 ry 50 rz -160.79 deg; joints [-8.613, -45.696, 108.75, 138.142, 69.263, 107.6, -289.206]
  MoveL 171 to (-55.59, 310.29, 0) mm, rotated rx -180 ry 50 rz 47.87 deg; joints [-20.194, -46.242, 111.219, 127.057, 74.288, 109.729, -137.87]
  Set speed (60.0 mm/s)
  MoveL 172 to (-37.62, 299.82, 0) mm, rotated rx 180 ry 50 rz 43.38 deg; joints [-20.194, -47.371, 111.315, 126.82, 73.668, 110.587, -133.377]
  MoveL 173 to (34.79, 183.72, 290) mm, rotated rx -180 ry 50 rz -155.49 deg; joints [-8.613, -44.618, 108.643, 138.382, 69.987, 106.912, -294.515]
  Set speed (60.0 mm/s)
  MoveL 174 to (31.73, 182.3, 280) mm, rotated rx 180 ry 50 rz -157.79 deg; joints [-9.003, -44.69, 108.816, 138.01, 70.176, 106.975, -292.214]
  MoveL 175 to (27.92, 180.74, 270) mm, rotated rx 180 ry 50 rz -160.59 deg; joints [-9.393, -44.76, 108.983, 137.637, 70.362, 107.039, -289.407]
  MoveL 176 to (23.38, 179.17, 260) mm, rotated rx 180 ry 50 rz -163.87 deg; joints [-9.784, -44.826, 109.144, 137.263, 70.547, 107.104, -286.13]
  MoveL 177 to (18.11, 177.74, 250) mm, rotated rx -180 ry 50 rz -167.58 deg; joints [-10.177, -44.89, 109.298, 136.887, 70.729, 107.171, -282.417]
  MoveL 178 to (12.17, 176.57, 240) mm, rotated rx 180 ry 50 rz -171.7 deg; joints [-10.57, -44.952, 109.447, 136.51, 70.908, 107.239, -278.3]
  MoveL 179 to (5.61, 175.83, 230) mm, rotated rx -180 ry 50 rz -176.19 deg; joints [-10.964, -45.013, 109.589, 136.131, 71.084, 107.309, -273.813]
  MoveL 180 to (-1.49, 175.64, 220) mm, rotated rx -180 ry 50 rz 178.99 deg; joints [-11.359, -45.073, 109.726, 135.751, 71.257, 107.381, -268.987]
  MoveL 181 to (-9.03, 176.15, 210) mm, rotated rx -180 ry 50 rz 173.85 deg; joints [-11.755, -45.133, 109.856, 135.369, 71.426, 107.456, -263.854]
  MoveL 182 to (-16.88, 177.46, 200) mm, rotated rx 180 ry 50 rz 168.44 deg; joints [-12.152, -45.193, 109.981, 134.985, 71.591, 107.535, -258.444]
  MoveL 183 to (-24.89, 179.66, 190) mm, rotated rx 180 ry 50 rz 162.78 deg; joints [-12.549, -45.254, 110.1, 134.6, 71.752, 107.617, -252.785]
  MoveL 184 to (-32.91, 182.83, 180) mm, rotated rx -180 ry 50 rz 156.91 deg; joints [-12.947, -45.316, 110.213, 134.212, 71.909, 107.702, -246.906]
  MoveL 185 to (-40.75, 186.98, 170) mm, rotated rx -180 ry 50 rz 150.84 deg; joints [-13.346, -45.378, 110.321, 133.823, 72.062, 107.792, -240.836]
  MoveL 186 to (-48.24, 192.12, 160) mm, rotated rx 180 ry 50 rz 144.6 deg; joints [-13.746, -45.442, 110.422, 133.433, 72.21, 107.886, -234.602]
  MoveL 187 to (-55.2, 198.19, 150) mm, rotated rx -180 ry 50 rz 138.23 deg; joints [-14.146, -45.506, 110.518, 133.04, 72.355, 107.983, -228.231]
  MoveL 188 to (-61.48, 205.13, 140) mm, rotated rx -180 ry 50 rz 131.75 deg; joints [-14.546, -45.571, 110.608, 132.647, 72.496, 108.085, -221.752]
  MoveL 189 to (-66.92, 212.81, 130) mm, rotated rx 180 ry 50 rz 125.19 deg; joints [-14.948, -45.636, 110.692, 132.251, 72.634, 108.19, -215.192]
  MoveL 190 to (-71.41, 221.1, 120) mm, rotated rx -180 ry 50 rz 118.58 deg; joints [-15.349, -45.701, 110.77, 131.855, 72.768, 108.299, -208.581]
  MoveL 191 to (-74.87, 229.83, 110) mm, rotated rx 180 ry 50 rz 111.95 deg; joints [-15.751, -45.765, 110.842, 131.457, 72.9, 108.41, -201.949]
  MoveL 192 to (-77.24, 238.83, 100) mm, rotated rx 180 ry 50 rz 105.33 deg; joints [-16.154, -45.828, 110.908, 131.058, 73.03, 108.525, -195.327]
  MoveL 193 to (-78.53, 247.91, 90) mm, rotated rx -180 ry 50 rz 98.75 deg; joints [-16.557, -45.889, 110.968, 130.659, 73.157, 108.642, -188.75]
  MoveL 194 to (-78.77, 256.9, 80) mm, rotated rx -180 ry 50 rz 92.25 deg; joints [-16.96, -45.947, 111.022, 130.259, 73.284, 108.76, -182.251]
  MoveL 195 to (-78, 265.63, 70) mm, rotated rx -180 ry 50 rz 85.87 deg; joints [-17.364, -46.001, 111.069, 129.859, 73.41, 108.88, -175.868]
  MoveL 196 to (-76.35, 273.96, 60) mm, rotated rx 180 ry 50 rz 79.64 deg; joints [-17.768, -46.051, 111.11, 129.458, 73.535, 109.001, -169.641]
  MoveL 197 to (-73.92, 281.75, 50) mm, rotated rx -180 ry 50 rz 73.61 deg; joints [-18.172, -46.097, 111.144, 129.057, 73.66, 109.122, -163.608]
  MoveL 198 to (-70.87, 288.9, 40) mm, rotated rx -180 ry 50 rz 67.81 deg; joints [-18.576, -46.137, 111.172, 128.657, 73.785, 109.244, -157.812]
  MoveL 199 to (-67.34, 295.36, 30) mm, rotated rx 180 ry 50 rz 62.3 deg; joints [-18.981, -46.172, 111.194, 128.256, 73.91, 109.365, -152.296]
  MoveL 200 to (-63.51, 301.08, 20) mm, rotated rx 180 ry 50 rz 57.1 deg; joints [-19.385, -46.201, 111.208, 127.856, 74.036, 109.487, -147.105]
  MoveL 201 to (-59.54, 306.05, 10) mm, rotated rx 180 ry 50 rz 52.28 deg; joints [-19.79, -46.225, 111.217, 127.456, 74.162, 109.608, -142.281]
  MoveL 202 to (-55.59, 310.29, 0) mm, rotated rx 180 ry 50 rz 47.87 deg; joints [-20.194, -46.242, 111.219, 127.057, 74.288, 109.729, -137.87]
  MoveL 203 to (34.79, 183.72, 290) mm, rotated rx -180 ry 50 rz -155.49 deg; joints [-8.613, -44.618, 108.643, 138.382, 69.987, 106.912, -294.515]
  Set speed (60.0 mm/s)
  MoveL 204 to (30.72, 204.12, 290) mm, rotated rx -180 ry 50 rz -151.2 deg; joints [-8.613, -45.718, 108.752, 138.137, 69.248, 107.615, -298.796]
  MoveL 205 to (-55.59, 310.29, 0) mm, rotated rx -180 ry 50 rz 47.87 deg; joints [-20.194, -46.242, 111.219, 127.057, 74.288, 109.729, -137.87]
  Set speed (60.0 mm/s)
  MoveL 206 to (-45.21, 292.27, 0) mm, rotated rx -180 ry 50 rz 54.48 deg; joints [-20.194, -47.328, 111.312, 126.829, 73.692, 110.554, -144.484]
  MoveL 207 to (-55.59, 310.29, 0) mm, rotated rx -180 ry 50 rz 47.87 deg; joints [-20.194, -46.242, 111.219, 127.057, 74.288, 109.729, -137.87]
  Set speed (60.0 mm/s)
  MoveL 208 to (-59.54, 306.05, 10) mm, rotated rx 180 ry 50 rz 52.28 deg; joints [-19.79, -46.225, 111.217, 127.456, 74.162, 109.608, -142.281]
  MoveL 209 to (-63.51, 301.08, 20) mm, rotated rx -180 ry 50 rz 57.1 deg; joints [-19.385, -46.201, 111.208, 127.856, 74.036, 109.487, -147.105]
  MoveL 210 to (-67.34, 295.36, 30) mm, rotated rx 180 ry 50 rz 62.3 deg; joints [-18.981, -46.172, 111.194, 128.256, 73.91, 109.365, -152.296]
  MoveL 211 to (-70.87, 288.9, 40) mm, rotated rx 180 ry 50 rz 67.81 deg; joints [-18.576, -46.137, 111.172, 128.657, 73.785, 109.244, -157.812]
  MoveL 212 to (-73.92, 281.75, 50) mm, rotated rx -180 ry 50 rz 73.61 deg; joints [-18.172, -46.097, 111.144, 129.057, 73.66, 109.122, -163.608]
  MoveL 213 to (-76.35, 273.96, 60) mm, rotated rx -180 ry 50 rz 79.64 deg; joints [-17.768, -46.051, 111.11, 129.458, 73.535, 109.001, -169.641]
  MoveL 214 to (-78, 265.63, 70) mm, rotated rx -180 ry 50 rz 85.87 deg; joints [-17.364, -46.001, 111.069, 129.859, 73.41, 108.88, -175.868]
  MoveL 215 to (-78.77, 256.9, 80) mm, rotated rx 180 ry 50 rz 92.25 deg; joints [-16.96, -45.947, 111.022, 130.259, 73.284, 108.76, -182.251]
  MoveL 216 to (-78.53, 247.91, 90) mm, rotated rx 180 ry 50 rz 98.75 deg; joints [-16.557, -45.889, 110.968, 130.659, 73.157, 108.642, -188.75]
  MoveL 217 to (-77.24, 238.83, 100) mm, rotated rx 180 ry 50 rz 105.33 deg; joints [-16.154, -45.828, 110.908, 131.058, 73.03, 108.525, -195.327]
  MoveL 218 to (-74.87, 229.83, 110) mm, rotated rx 180 ry 50 rz 111.95 deg; joints [-15.751, -45.765, 110.842, 131.457, 72.9, 108.41, -201.949]
  MoveL 219 to (-71.41, 221.1, 120) mm, rotated rx -180 ry 50 rz 118.58 deg; joints [-15.349, -45.701, 110.77, 131.855, 72.768, 108.299, -208.581]
  MoveL 220 to (-66.92, 212.81, 130) mm, rotated rx -180 ry 50 rz 125.19 deg; joints [-14.948, -45.636, 110.692, 132.251, 72.634, 108.19, -215.192]
  MoveL 221 to (-61.48, 205.13, 140) mm, rotated rx 180 ry 50 rz 131.75 deg; joints [-14.546, -45.571, 110.608, 132.647, 72.496, 108.085, -221.752]
  MoveL 222 to (-55.2, 198.19, 150) mm, rotated rx -180 ry 50 rz 138.23 deg; joints [-14.146, -45.506, 110.518, 133.04, 72.355, 107.983, -228.231]
  MoveL 223 to (-48.24, 192.12, 160) mm, rotated rx 180 ry 50 rz 144.6 deg; joints [-13.746, -45.442, 110.422, 133.433, 72.21, 107.886, -234.602]
  MoveL 224 to (-40.75, 186.98, 170) mm, rotated rx 180 ry 50 rz 150.84 deg; joints [-13.346, -45.378, 110.321, 133.823, 72.062, 107.792, -240.836]
  MoveL 225 to (-32.91, 182.83, 180) mm, rotated rx 180 ry 50 rz 156.91 deg; joints [-12.947, -45.316, 110.213, 134.212, 71.909, 107.702, -246.906]
  MoveL 226 to (-24.89, 179.66, 190) mm, rotated rx -180 ry 50 rz 162.78 deg; joints [-12.549, -45.254, 110.1, 134.6, 71.752, 107.617, -252.785]
  MoveL 227 to (-16.88, 177.46, 200) mm, rotated rx -180 ry 50 rz 168.44 deg; joints [-12.152, -45.193, 109.981, 134.985, 71.591, 107.535, -258.444]
  MoveL 228 to (-9.03, 176.15, 210) mm, rotated rx -180 ry 50 rz 173.85 deg; joints [-11.755, -45.133, 109.856, 135.369, 71.426, 107.456, -263.854]
  MoveL 229 to (-1.49, 175.64, 220) mm, rotated rx -180 ry 50 rz 178.99 deg; joints [-11.359, -45.073, 109.726, 135.751, 71.257, 107.381, -268.987]
  MoveL 230 to (5.61, 175.83, 230) mm, rotated rx -180 ry 50 rz -176.19 deg; joints [-10.964, -45.013, 109.589, 136.131, 71.084, 107.309, -273.813]
  MoveL 231 to (12.17, 176.57, 240) mm, rotated rx 180 ry 50 rz -171.7 deg; joints [-10.57, -44.952, 109.447, 136.51, 70.908, 107.239, -278.3]
  MoveL 232 to (18.11, 177.74, 250) mm, rotated rx -180 ry 50 rz -167.58 deg; joints [-10.177, -44.89, 109.298, 136.887, 70.729, 107.171, -282.417]
  MoveL 233 to (23.38, 179.17, 260) mm, rotated rx -180 ry 50 rz -163.87 deg; joints [-9.784, -44.826, 109.144, 137.263, 70.547, 107.104, -286.13]
  MoveL 234 to (27.92, 180.74, 270) mm, rotated rx 180 ry 50 rz -160.59 deg; joints [-9.393, -44.76, 108.983, 137.637, 70.362, 107.039, -289.407]
  MoveL 235 to (31.73, 182.3, 280) mm, rotated rx 180 ry 50 rz -157.79 deg; joints [-9.003, -44.69, 108.816, 138.01, 70.176, 106.975, -292.214]
  MoveL 236 to (34.79, 183.72, 290) mm, rotated rx 180 ry 50 rz -155.49 deg; joints [-8.613, -44.618, 108.643, 138.382, 69.987, 106.912, -294.515]
  MoveL 237 to (30.72, 204.12, 290) mm, rotated rx 180 ry 50 rz -151.2 deg; joints [-8.613, -45.718, 108.752, 138.137, 69.248, 107.615, -298.796]
  Set speed (60.0 mm/s)
  MoveL 238 to (28.54, 202.85, 280) mm, rotated rx 180 ry 50 rz -153.47 deg; joints [-9.003, -45.792, 108.925, 137.765, 69.44, 107.683, -296.535]
  MoveL 239 to (25.81, 201.43, 270) mm, rotated rx -180 ry 50 rz -156.22 deg; joints [-9.393, -45.861, 109.092, 137.393, 69.631, 107.752, -293.779]
  MoveL 240 to (22.53, 199.96, 260) mm, rotated rx -180 ry 50 rz -159.44 deg; joints [-9.784, -45.928, 109.253, 137.019, 69.819, 107.822, -290.563]
  MoveL 241 to (18.7, 198.53, 250) mm, rotated rx 180 ry 50 rz -163.08 deg; joints [-10.177, -45.992, 109.408, 136.644, 70.006, 107.892, -286.921]
  MoveL 242 to (14.35, 197.26, 240) mm, rotated rx 180 ry 50 rz -167.11 deg; joints [-10.57, -46.054, 109.557, 136.268, 70.189, 107.965, -282.886]
  MoveL 243 to (9.52, 196.26, 230) mm, rotated rx 180 ry 50 rz -171.51 deg; joints [-10.964, -46.115, 109.699, 135.89, 70.37, 108.038, -278.492]
  MoveL 244 to (4.24, 195.64, 220) mm, rotated rx -180 ry 50 rz -176.23 deg; joints [-11.359, -46.174, 109.835, 135.511, 70.548, 108.115, -273.769]
  MoveL 245 to (-1.41, 195.5, 210) mm, rotated rx 180 ry 50 rz 178.75 deg; joints [-11.755, -46.233, 109.966, 135.13, 70.722, 108.194, -268.748]
  MoveL 246 to (-7.35, 195.94, 200) mm, rotated rx 180 ry 50 rz 173.46 deg; joints [-12.152, -46.292, 110.09, 134.747, 70.893, 108.276, -263.458]
  MoveL 247 to (-13.47, 197.04, 190) mm, rotated rx 180 ry 50 rz 167.93 deg; joints [-12.549, -46.351, 110.209, 134.362, 71.059, 108.361, -257.927]
  MoveL 248 to (-19.65, 198.85, 180) mm, rotated rx 180 ry 50 rz 162.18 deg; joints [-12.947, -46.411, 110.322, 133.976, 71.222, 108.45, -252.183]
  MoveL 249 to (-25.78, 201.42, 170) mm, rotated rx 180 ry 50 rz 156.25 deg; joints [-13.346, -46.471, 110.428, 133.588, 71.38, 108.542, -246.252]
  MoveL 250 to (-31.7, 204.73, 160) mm, rotated rx -180 ry 50 rz 150.16 deg; joints [-13.746, -46.533, 110.529, 133.198, 71.535, 108.639, -240.159]
  MoveL 251 to (-37.3, 208.79, 150) mm, rotated rx 180 ry 50 rz 143.93 deg; joints [-14.146, -46.595, 110.624, 132.807, 71.685, 108.74, -233.93]
  MoveL 252 to (-42.45, 213.53, 140) mm, rotated rx 180 ry 50 rz 137.59 deg; joints [-14.546, -46.658, 110.713, 132.414, 71.832, 108.845, -227.591]
  MoveL 253 to (-47.02, 218.88, 130) mm, rotated rx 180 ry 50 rz 131.17 deg; joints [-14.948, -46.721, 110.796, 132.019, 71.975, 108.953, -221.168]
  MoveL 254 to (-50.93, 224.75, 120) mm, rotated rx 180 ry 50 rz 124.69 deg; joints [-15.349, -46.784, 110.873, 131.623, 72.115, 109.066, -214.687]
  MoveL 255 to (-54.1, 231.02, 110) mm, rotated rx 180 ry 50 rz 118.18 deg; joints [-15.751, -46.847, 110.944, 131.226, 72.253, 109.181, -208.176]
  MoveL 256 to (-56.49, 237.56, 100) mm, rotated rx 180 ry 50 rz 111.66 deg; joints [-16.154, -46.909, 111.009, 130.828, 72.388, 109.3, -201.664]
  MoveL 257 to (-58.06, 244.24, 90) mm, rotated rx -180 ry 50 rz 105.18 deg; joints [-16.557, -46.968, 111.068, 130.429, 72.52, 109.421, -195.184]
  MoveL 258 to (-58.85, 250.92, 80) mm, rotated rx 180 ry 50 rz 98.77 deg; joints [-16.96, -47.026, 111.12, 130.029, 72.652, 109.544, -188.767]
  MoveL 259 to (-58.87, 257.48, 70) mm, rotated rx 180 ry 50 rz 92.45 deg; joints [-17.364, -47.08, 111.167, 129.629, 72.782, 109.669, -182.451]
  MoveL 260 to (-58.2, 263.79, 60) mm, rotated rx 180 ry 50 rz 86.27 deg; joints [-17.768, -47.13, 111.206, 129.229, 72.912, 109.795, -176.272]
  MoveL 261 to (-56.92, 269.76, 50) mm, rotated rx 180 ry 50 rz 80.27 deg; joints [-18.172, -47.177, 111.24, 128.829, 73.041, 109.921, -170.271]
  MoveL 262 to (-55.13, 275.3, 40) mm, rotated rx 180 ry 50 rz 74.49 deg; joints [-18.576, -47.218, 111.267, 128.428, 73.171, 110.048, -164.491]
  MoveL 263 to (-52.95, 280.35, 30) mm, rotated rx 180 ry 50 rz 68.98 deg; joints [-18.981, -47.254, 111.288, 128.028, 73.3, 110.175, -158.976]
  MoveL 264 to (-50.48, 284.87, 20) mm, rotated rx 180 ry 50 rz 63.77 deg; joints [-19.385, -47.284, 111.302, 127.628, 73.43, 110.302, -153.772]
  MoveL 265 to (-47.86, 288.84, 10) mm, rotated rx 180 ry 50 rz 58.93 deg; joints [-19.79, -47.309, 111.31, 127.228, 73.561, 110.428, -148.926]
  MoveL 266 to (-45.21, 292.27, 0) mm, rotated rx 180 ry 50 rz 54.48 deg; joints [-20.194, -47.328, 111.312, 126.829, 73.692, 110.554, -144.484]
  MoveL 267 to (30.72, 204.12, 290) mm, rotated rx -180 ry 50 rz -151.2 deg; joints [-8.613, -45.718, 108.752, 138.137, 69.248, 107.615, -298.796]
  Set speed (60.0 mm/s)
  MoveL 268 to (58.22, 245.2, 290) mm, rotated rx -180 ry 50 rz -104.27 deg; joints [-8.613, -45.919, 108.769, 138.09, 69.111, 107.747, -345.735]
  MoveL 269 to (-45.21, 292.27, 0) mm, rotated rx 180 ry 50 rz 54.48 deg; joints [-20.194, -47.328, 111.312, 126.829, 73.692, 110.554, -504.484]
  Set speed (60.0 mm/s)
  MoveL 270 to (-58.12, 244.54, 0) mm, rotated rx -180 ry 50 rz 104.89 deg; joints [-20.194, -47.073, 111.293, 126.884, 73.834, 110.357, -554.894]
  MoveL 271 to (-45.21, 292.27, 0) mm, rotated rx 180 ry 50 rz 54.48 deg; joints [-20.194, -47.328, 111.312, 126.829, 73.692, 110.554, -504.484]
  Set speed (60.0 mm/s)
  MoveL 272 to (-47.86, 288.84, 10) mm, rotated rx 180 ry 50 rz 58.93 deg; joints [-19.79, -47.309, 111.31, 127.228, 73.561, 110.428, -508.926]
  MoveL 273 to (-50.48, 284.87, 20) mm, rotated rx 180 ry 50 rz 63.77 deg; joints [-19.385, -47.284, 111.302, 127.628, 73.43, 110.302, -513.772]
  MoveL 274 to (-52.95, 280.35, 30) mm, rotated rx 180 ry 50 rz 68.98 deg; joints [-18.981, -47.254, 111.288, 128.028, 73.3, 110.175, -518.976]
  MoveL 275 to (-55.13, 275.3, 40) mm, rotated rx -180 ry 50 rz 74.49 deg; joints [-18.576, -47.218, 111.267, 128.428, 73.171, 110.048, -524.491]
  MoveL 276 to (-56.92, 269.76, 50) mm, rotated rx 180 ry 50 rz 80.27 deg; joints [-18.172, -47.177, 111.24, 128.829, 73.041, 109.921, -530.271]
  MoveL 277 to (-58.2, 263.79, 60) mm, rotated rx 180 ry 50 rz 86.27 deg; joints [-17.768, -47.13, 111.206, 129.229, 72.912, 109.795, -536.272]
  MoveL 278 to (-58.87, 257.48, 70) mm, rotated rx 180 ry 50 rz 92.45 deg; joints [-17.364, -47.08, 111.167, 129.629, 72.782, 109.669, -542.451]
  MoveL 279 to (-58.85, 250.92, 80) mm, rotated rx 180 ry 50 rz 98.77 deg; joints [-16.96, -47.026, 111.12, 130.029, 72.652, 109.544, -548.767]
  MoveL 280 to (-58.06, 244.24, 90) mm, rotated rx 180 ry 50 rz 105.18 deg; joints [-16.557, -46.968, 111.068, 130.429, 72.52, 109.421, -555.184]
  MoveL 281 to (-56.49, 237.56, 100) mm, rotated rx 180 ry 50 rz 111.66 deg; joints [-16.154, -46.909, 111.009, 130.828, 72.388, 109.3, -561.664]
  MoveL 282 to (-54.1, 231.02, 110) mm, rotated rx 180 ry 50 rz 118.18 deg; joints [-15.751, -46.847, 110.944, 131.226, 72.253, 109.181, -568.176]
  MoveL 283 to (-50.93, 224.75, 120) mm, rotated rx -180 ry 50 rz 124.69 deg; joints [-15.349, -46.784, 110.873, 131.623, 72.115, 109.066, -574.687]
  MoveL 284 to (-47.02, 218.88, 130) mm, rotated rx -180 ry 50 rz 131.17 deg; joints [-14.948, -46.721, 110.796, 132.019, 71.975, 108.953, -581.168]
  MoveL 285 to (-42.45, 213.53, 140) mm, rotated rx -180 ry 50 rz 137.59 deg; joints [-14.546, -46.658, 110.713, 132.414, 71.832, 108.845, -587.591]
  MoveL 286 to (-37.3, 208.79, 150) mm, rotated rx -180 ry 50 rz 143.93 deg; joints [-14.146, -46.595, 110.624, 132.807, 71.685, 108.74, -593.93]
  MoveL 287 to (-31.7, 204.73, 160) mm, rotated rx 180 ry 50 rz 150.16 deg; joints [-13.746, -46.533, 110.529, 133.198, 71.535, 108.639, -600.159]
  MoveL 288 to (-25.78, 201.42, 170) mm, rotated rx 180 ry 50 rz 156.25 deg; joints [-13.346, -46.471, 110.428, 133.588, 71.38, 108.542, -606.252]
  MoveL 289 to (-19.65, 198.85, 180) mm, rotated rx 180 ry 50 rz 162.18 deg; joints [-12.947, -46.411, 110.322, 133.976, 71.222, 108.45, -612.183]
  MoveL 290 to (-13.47, 197.04, 190) mm, rotated rx 180 ry 50 rz 167.93 deg; joints [-12.549, -46.351, 110.209, 134.362, 71.059, 108.361, -617.927]
  MoveL 291 to (-7.35, 195.94, 200) mm, rotated rx 180 ry 50 rz 173.46 deg; joints [-12.152, -46.292, 110.09, 134.747, 70.893, 108.276, -623.458]
  MoveL 292 to (-1.41, 195.5, 210) mm, rotated rx -180 ry 50 rz 178.75 deg; joints [-11.755, -46.233, 109.966, 135.13, 70.722, 108.194, -628.748]
  MoveL 293 to (4.24, 195.64, 220) mm, rotated rx -180 ry 50 rz -176.23 deg; joints [-11.359, -46.174, 109.835, 135.511, 70.548, 108.115, -633.769]
  MoveL 294 to (9.52, 196.26, 230) mm, rotated rx -180 ry 50 rz -171.51 deg; joints [-10.964, -46.115, 109.699, 135.89, 70.37, 108.038, -638.492]
  MoveL 295 to (14.35, 197.26, 240) mm, rotated rx 180 ry 50 rz -167.11 deg; joints [-10.57, -46.054, 109.557, 136.268, 70.189, 107.965, -642.886]
  MoveL 296 to (18.7, 198.53, 250) mm, rotated rx 180 ry 50 rz -163.08 deg; joints [-10.177, -45.992, 109.408, 136.644, 70.006, 107.892, -646.921]
  MoveL 297 to (22.53, 199.96, 260) mm, rotated rx -180 ry 50 rz -159.44 deg; joints [-9.784, -45.928, 109.253, 137.019, 69.819, 107.822, -650.563]
  MoveL 298 to (25.81, 201.43, 270) mm, rotated rx 180 ry 50 rz -156.22 deg; joints [-9.393, -45.861, 109.092, 137.393, 69.631, 107.752, -653.779]
  MoveL 299 to (28.54, 202.85, 280) mm, rotated rx 180 ry 50 rz -153.47 deg; joints [-9.003, -45.792, 108.925, 137.765, 69.44, 107.683, -656.535]
  MoveL 300 to (30.72, 204.12, 290) mm, rotated rx 180 ry 50 rz -151.2 deg; joints [-8.613, -45.718, 108.752, 138.137, 69.248, 107.615, -658.796]
  MoveL 301 to (58.22, 245.2, 290) mm, rotated rx -180 ry 50 rz -104.27 deg; joints [-8.613, -45.919, 108.769, 138.09, 69.111, 107.747, -705.735]
  Set speed (60.0 mm/s)
  MoveL 302 to (57.77, 242.72, 280) mm, rotated rx -180 ry 50 rz -106.66 deg; joints [-9.003, -45.986, 108.941, 137.72, 69.308, 107.812, -703.345]
  MoveL 303 to (57.08, 239.72, 270) mm, rotated rx -180 ry 50 rz -109.56 deg; joints [-9.393, -46.048, 109.108, 137.35, 69.505, 107.876, -700.439]
  MoveL 304 to (56.08, 236.26, 260) mm, rotated rx 180 ry 50 rz -112.94 deg; joints [-9.784, -46.105, 109.268, 136.978, 69.701, 107.94, -697.057]
  MoveL 305 to (54.69, 232.42, 250) mm, rotated rx -180 ry 50 rz -116.76 deg; joints [-10.177, -46.157, 109.422, 136.606, 69.896, 108.003, -693.242]
  MoveL 306 to (52.84, 228.29, 240) mm, rotated rx -180 ry 50 rz -120.97 deg; joints [-10.57, -46.205, 109.569, 136.233, 70.09, 108.066, -689.031]
  MoveL 307 to (50.46, 223.96, 230) mm, rotated rx -180 ry 50 rz -125.53 deg; joints [-10.964, -46.249, 109.71, 135.859, 70.282, 108.129, -684.466]
  MoveL 308 to (47.51, 219.54, 220) mm, rotated rx -180 ry 50 rz -130.42 deg; joints [-11.359, -46.29, 109.845, 135.484, 70.473, 108.193, -679.584]
  MoveL 309 to (43.95, 215.15, 210) mm, rotated rx 180 ry 50 rz -135.58 deg; joints [-11.755, -46.328, 109.974, 135.108, 70.661, 108.258, -674.422]
  MoveL 310 to (39.77, 210.92, 200) mm, rotated rx 180 ry 50 rz -140.98 deg; joints [-12.152, -46.364, 110.096, 134.731, 70.846, 108.325, -669.016]
  MoveL 311 to (34.96, 206.97, 190) mm, rotated rx 180 ry 50 rz -146.6 deg; joints [-12.549, -46.399, 110.213, 134.352, 71.029, 108.394, -663.399]
  MoveL 312 to (29.57, 203.44, 180) mm, rotated rx 180 ry 50 rz -152.4 deg; joints [-12.947, -46.433, 110.323, 133.971, 71.208, 108.465, -657.602]
  MoveL 313 to (23.65, 200.44, 170) mm, rotated rx 180 ry 50 rz -158.34 deg; joints [-13.346, -46.467, 110.428, 133.589, 71.383, 108.539, -651.658]
  MoveL 314 to (17.28, 198.07, 160) mm, rotated rx -180 ry 50 rz -164.41 deg; joints [-13.746, -46.501, 110.526, 133.205, 71.555, 108.617, -645.594]
  MoveL 315 to (10.57, 196.44, 150) mm, rotated rx -180 ry 50 rz -170.56 deg; joints [-14.146, -46.535, 110.619, 132.82, 71.723, 108.698, -639.438]
  MoveL 316 to (3.62, 195.59, 140) mm, rotated rx 180 ry 50 rz -176.78 deg; joints [-14.546, -46.571, 110.706, 132.433, 71.886, 108.783, -633.219]
  MoveL 317 to (-3.42, 195.58, 130) mm, rotated rx 180 ry 50 rz 176.96 deg; joints [-14.948, -46.607, 110.787, 132.044, 72.045, 108.872, -626.961]
  MoveL 318 to (-10.42, 196.41, 120) mm, rotated rx -180 ry 50 rz 170.69 deg; joints [-15.349, -46.645, 110.862, 131.654, 72.2, 108.966, -620.691]
  MoveL 319 to (-17.25, 198.06, 110) mm, rotated rx -180 ry 50 rz 164.44 deg; joints [-15.751, -46.685, 110.931, 131.262, 72.351, 109.064, -614.435]
  MoveL 320 to (-23.78, 200.49, 100) mm, rotated rx -180 ry 50 rz 158.22 deg; joints [-16.154, -46.725, 110.994, 130.869, 72.498, 109.166, -608.22]
  MoveL 321 to (-29.89, 203.62, 90) mm, rotated rx -180 ry 50 rz 152.07 deg; joints [-16.557, -46.765, 111.051, 130.474, 72.641, 109.272, -602.072]
  MoveL 322 to (-35.48, 207.36, 80) mm, rotated rx 180 ry 50 rz 146.02 deg; joints [-16.96, -46.806, 111.103, 130.078, 72.782, 109.382, -596.02]
  MoveL 323 to (-40.49, 211.59, 70) mm, rotated rx -180 ry 50 rz 140.09 deg; joints [-17.364, -46.847, 111.148, 129.68, 72.919, 109.496, -590.093]
  MoveL 324 to (-44.86, 216.19, 60) mm, rotated rx 180 ry 50 rz 134.32 deg; joints [-17.768, -46.887, 111.187, 129.282, 73.054, 109.613, -584.321]
  MoveL 325 to (-48.58, 221.03, 50) mm, rotated rx -180 ry 50 rz 128.74 deg; joints [-18.172, -46.925, 111.22, 128.883, 73.187, 109.732, -578.737]
  MoveL 326 to (-51.63, 225.99, 40) mm, rotated rx 180 ry 50 rz 123.38 deg; joints [-18.576, -46.961, 111.247, 128.484, 73.318, 109.854, -573.376]
  MoveL 327 to (-54.06, 230.92, 30) mm, rotated rx 180 ry 50 rz 118.27 deg; joints [-18.981, -46.994, 111.268, 128.084, 73.448, 109.978, -568.272]
  MoveL 328 to (-55.91, 235.73, 20) mm, rotated rx 180 ry 50 rz 113.46 deg; joints [-19.385, -47.025, 111.283, 127.684, 73.577, 110.103, -563.465]
  MoveL 329 to (-57.23, 240.3, 10) mm, rotated rx 180 ry 50 rz 108.99 deg; joints [-19.79, -47.051, 111.291, 127.284, 73.705, 110.23, -558.992]
  MoveL 330 to (-58.12, 244.54, 0) mm, rotated rx 180 ry 50 rz 104.89 deg; joints [-20.194, -47.073, 111.293, 126.884, 73.834, 110.357, -554.894]
  MoveL 331 to (58.22, 245.2, 290) mm, rotated rx -180 ry 50 rz -104.27 deg; joints [-8.613, -45.919, 108.769, 138.09, 69.111, 107.747, -705.735]
  Set speed (60.0 mm/s)
  MoveL 332 to (78.63, 249.2, 290) mm, rotated rx -180 ry 50 rz -97.82 deg; joints [-8.613, -44.864, 108.67, 138.329, 69.824, 107.066, -712.181]
  MoveL 333 to (-58.12, 244.54, 0) mm, rotated rx 180 ry 50 rz 104.89 deg; joints [-20.194, -47.073, 111.293, 126.884, 73.834, 110.357, -554.894]
  Set speed (60.0 mm/s)
  MoveL 334 to (-76.17, 234.21, 0) mm, rotated rx 180 ry 50 rz 108.7 deg; joints [-20.194, -45.935, 111.187, 127.118, 74.455, 109.5, -558.703]
  MoveL 335 to (-58.12, 244.54, 0) mm, rotated rx 180 ry 50 rz 104.89 deg; joints [-20.194, -47.073, 111.293, 126.884, 73.834, 110.357, -554.894]
  Set speed (60.0 mm/s)
  MoveL 336 to (-57.23, 240.3, 10) mm, rotated rx 180 ry 50 rz 108.99 deg; joints [-19.79, -47.051, 111.291, 127.284, 73.705, 110.23, -558.992]
  MoveL 337 to (-55.91, 235.73, 20) mm, rotated rx -180 ry 50 rz 113.46 deg; joints [-19.385, -47.025, 111.283, 127.684, 73.577, 110.103, -563.465]
  MoveL 338 to (-54.06, 230.92, 30) mm, rotated rx 180 ry 50 rz 118.27 deg; joints [-18.981, -46.994, 111.268, 128.084, 73.448, 109.978, -568.272]
  MoveL 339 to (-51.63, 225.99, 40) mm, rotated rx 180 ry 50 rz 123.38 deg; joints [-18.576, -46.961, 111.247, 128.484, 73.318, 109.854, -573.376]
  MoveL 340 to (-48.58, 221.03, 50) mm, rotated rx 180 ry 50 rz 128.74 deg; joints [-18.172, -46.925, 111.22, 128.883, 73.187, 109.732, -578.737]
  MoveL 341 to (-44.86, 216.19, 60) mm, rotated rx 180 ry 50 rz 134.32 deg; joints [-17.768, -46.887, 111.187, 129.282, 73.054, 109.613, -584.321]
  MoveL 342 to (-40.49, 211.59, 70) mm, rotated rx 180 ry 50 rz 140.09 deg; joints [-17.364, -46.847, 111.148, 129.68, 72.919, 109.496, -590.093]
  MoveL 343 to (-35.48, 207.36, 80) mm, rotated rx -180 ry 50 rz 146.02 deg; joints [-16.96, -46.806, 111.103, 130.078, 72.782, 109.382, -596.02]
  MoveL 344 to (-29.89, 203.62, 90) mm, rotated rx 180 ry 50 rz 152.07 deg; joints [-16.557, -46.765, 111.051, 130.474, 72.641, 109.272, -602.072]
  MoveL 345 to (-23.78, 200.49, 100) mm, rotated rx -180 ry 50 rz 158.22 deg; joints [-16.154, -46.725, 110.994, 130.869, 72.498, 109.166, -608.22]
  MoveL 346 to (-17.25, 198.06, 110) mm, rotated rx 180 ry 50 rz 164.44 deg; joints [-15.751, -46.685, 110.931, 131.262, 72.351, 109.064, -614.435]
  MoveL 347 to (-10.42, 196.41, 120) mm, rotated rx -180 ry 50 rz 170.69 deg; joints [-15.349, -46.645, 110.862, 131.654, 72.2, 108.966, -620.691]
  MoveL 348 to (-3.42, 195.58, 130) mm, rotated rx -180 ry 50 rz 176.96 deg; joints [-14.948, -46.607, 110.787, 132.044, 72.045, 108.872, -626.961]
  MoveL 349 to (3.62, 195.59, 140) mm, rotated rx 180 ry 50 rz -176.78 deg; joints [-14.546, -46.571, 110.706, 132.433, 71.886, 108.783, -633.219]
  MoveL 350 to (10.57, 196.44, 150) mm, rotated rx 180 ry 50 rz -170.56 deg; joints [-14.146, -46.535, 110.619, 132.82, 71.723, 108.698, -639.438]
  MoveL 351 to (17.28, 198.07, 160) mm, rotated rx -180 ry 50 rz -164.41 deg; joints [-13.746, -46.501, 110.526, 133.205, 71.555, 108.617, -645.594]
  MoveL 352 to (23.65, 200.44, 170) mm, rotated rx -180 ry 50 rz -158.34 deg; joints [-13.346, -46.467, 110.428, 133.589, 71.383, 108.539, -651.658]
  MoveL 353 to (29.57, 203.44, 180) mm, rotated rx 180 ry 50 rz -152.4 deg; joints [-12.947, -46.433, 110.323, 133.971, 71.208, 108.465, -657.602]
  MoveL 354 to (34.96, 206.97, 190) mm, rotated rx 180 ry 50 rz -146.6 deg; joints [-12.549, -46.399, 110.213, 134.352, 71.029, 108.394, -663.399]
  MoveL 355 to (39.77, 210.92, 200) mm, rotated rx 180 ry 50 rz -140.98 deg; joints [-12.152, -46.364, 110.096, 134.731, 70.846, 108.325, -669.016]
  MoveL 356 to (43.95, 215.15, 210) mm, rotated rx 180 ry 50 rz -135.58 deg; joints [-11.755, -46.328, 109.974, 135.108, 70.661, 108.258, -674.422]
  MoveL 357 to (47.51, 219.54, 220) mm, rotated rx 180 ry 50 rz -130.42 deg; joints [-11.359, -46.29, 109.845, 135.484, 70.473, 108.193, -679.584]
  MoveL 358 to (50.46, 223.96, 230) mm, rotated rx -180 ry 50 rz -125.53 deg; joints [-10.964, -46.249, 109.71, 135.859, 70.282, 108.129, -684.466]
  MoveL 359 to (52.84, 228.29, 240) mm, rotated rx -180 ry 50 rz -120.97 deg; joints [-10.57, -46.205, 109.569, 136.233, 70.09, 108.066, -689.031]
  MoveL 360 to (54.69, 232.42, 250) mm, rotated rx -180 ry 50 rz -116.76 deg; joints [-10.177, -46.157, 109.422, 136.606, 69.896, 108.003, -693.242]
  MoveL 361 to (56.08, 236.26, 260) mm, rotated rx -180 ry 50 rz -112.94 deg; joints [-9.784, -46.105, 109.268, 136.978, 69.701, 107.94, -697.057]
  MoveL 362 to (57.08, 239.72, 270) mm, rotated rx 180 ry 50 rz -109.56 deg; joints [-9.393, -46.048, 109.108, 137.35, 69.505, 107.876, -700.439]
  MoveL 363 to (57.77, 242.72, 280) mm, rotated rx -180 ry 50 rz -106.66 deg; joints [-9.003, -45.986, 108.941, 137.72, 69.308, 107.812, -703.345]
  MoveL 364 to (58.22, 245.2, 290) mm, rotated rx -180 ry 50 rz -104.27 deg; joints [-8.613, -45.919, 108.769, 138.09, 69.111, 107.747, -705.735]
  MoveL 365 to (78.63, 249.2, 290) mm, rotated rx -180 ry 50 rz -97.82 deg; joints [-8.613, -44.864, 108.67, 138.329, 69.824, 107.066, -712.181]
  Set speed (60.0 mm/s)
  MoveL 366 to (78.34, 245.85, 280) mm, rotated rx 180 ry 50 rz -100.24 deg; joints [-9.003, -44.929, 108.842, 137.958, 70.018, 107.126, -709.758]
  MoveL 367 to (77.78, 241.77, 270) mm, rotated rx -180 ry 50 rz -103.19 deg; joints [-9.393, -44.989, 109.008, 137.588, 70.212, 107.185, -706.809]
  MoveL 368 to (76.86, 237.05, 260) mm, rotated rx 180 ry 50 rz -106.63 deg; joints [-9.784, -45.043, 109.168, 137.216, 70.405, 107.243, -703.374]
  MoveL 369 to (75.48, 231.77, 250) mm, rotated rx -180 ry 50 rz -110.51 deg; joints [-10.177, -45.092, 109.321, 136.844, 70.597, 107.301, -699.493]
  MoveL 370 to (73.51, 226.04, 240) mm, rotated rx 180 ry 50 rz -114.79 deg; joints [-10.57, -45.137, 109.467, 136.47, 70.789, 107.358, -695.208]
  MoveL 371 to (70.88, 219.99, 230) mm, rotated rx -180 ry 50 rz -119.44 deg; joints [-10.964, -45.178, 109.608, 136.096, 70.978, 107.416, -690.555]
  MoveL 372 to (67.49, 213.75, 220) mm, rotated rx 180 ry 50 rz -124.42 deg; joints [-11.359, -45.216, 109.742, 135.721, 71.166, 107.474, -685.575]
  MoveL 373 to (63.28, 207.47, 210) mm, rotated rx 180 ry 50 rz -129.69 deg; joints [-11.755, -45.25, 109.87, 135.344, 71.352, 107.533, -680.305]
  MoveL 374 to (58.22, 201.33, 200) mm, rotated rx -180 ry 50 rz -135.22 deg; joints [-12.152, -45.282, 109.991, 134.966, 71.535, 107.594, -674.781]
  MoveL 375 to (52.31, 195.49, 190) mm, rotated rx 180 ry 50 rz -140.96 deg; joints [-12.549, -45.313, 110.107, 134.587, 71.715, 107.656, -669.037]
  MoveL 376 to (45.56, 190.13, 180) mm, rotated rx -180 ry 50 rz -146.89 deg; joints [-12.947, -45.343, 110.216, 134.207, 71.892, 107.721, -663.107]
  MoveL 377 to (38.04, 185.42, 170) mm, rotated rx -180 ry 50 rz -152.98 deg; joints [-13.346, -45.372, 110.32, 133.825, 72.065, 107.788, -657.024]
  MoveL 378 to (29.85, 181.5, 160) mm, rotated rx 180 ry 50 rz -159.18 deg; joints [-13.746, -45.402, 110.418, 133.441, 72.234, 107.859, -650.818]
  MoveL 379 to (21.11, 178.51, 150) mm, rotated rx 180 ry 50 rz -165.48 deg; joints [-14.146, -45.432, 110.51, 133.056, 72.4, 107.933, -644.519]
  MoveL 380 to (11.96, 176.54, 140) mm, rotated rx -180 ry 50 rz -171.84 deg; joints [-14.546, -45.464, 110.596, 132.669, 72.561, 108.011, -638.157]
  MoveL 381 to (2.59, 175.67, 130) mm, rotated rx 180 ry 50 rz -178.24 deg; joints [-14.948, -45.496, 110.677, 132.28, 72.717, 108.093, -631.758]
  MoveL 382 to (-6.83, 175.92, 120) mm, rotated rx 180 ry 50 rz 175.35 deg; joints [-15.349, -45.53, 110.751, 131.89, 72.869, 108.18, -625.352]
  MoveL 383 to (-16.13, 177.3, 110) mm, rotated rx -180 ry 50 rz 168.97 deg; joints [-15.751, -45.566, 110.82, 131.498, 73.018, 108.271, -618.967]
  MoveL 384 to (-25.11, 179.73, 100) mm, rotated rx 180 ry 50 rz 162.63 deg; joints [-16.154, -45.602, 110.884, 131.105, 73.162, 108.366, -612.629]
  MoveL 385 to (-33.62, 183.16, 90) mm, rotated rx 180 ry 50 rz 156.37 deg; joints [-16.557, -45.64, 110.941, 130.71, 73.302, 108.466, -606.369]
  MoveL 386 to (-41.52, 187.45, 80) mm, rotated rx -180 ry 50 rz 150.21 deg; joints [-16.96, -45.678, 110.993, 130.314, 73.439, 108.57, -600.214]
  MoveL 387 to (-48.7, 192.48, 70) mm, rotated rx 180 ry 50 rz 144.2 deg; joints [-17.364, -45.717, 111.038, 129.916, 73.572, 108.677, -594.197]
  MoveL 388 to (-55.08, 198.08, 60) mm, rotated rx -180 ry 50 rz 138.35 deg; joints [-17.768, -45.754, 111.078, 129.518, 73.703, 108.788, -588.347]
  MoveL 389 to (-60.61, 204.07, 50) mm, rotated rx -180 ry 50 rz 132.7 deg; joints [-18.172, -45.791, 111.112, 129.119, 73.832, 108.901, -582.698]
  MoveL 390 to (-65.29, 210.3, 40) mm, rotated rx -180 ry 50 rz 127.28 deg; joints [-18.576, -45.826, 111.139, 128.72, 73.959, 109.018, -577.284]
  MoveL 391 to (-69.12, 216.58, 30) mm, rotated rx -180 ry 50 rz 122.14 deg; joints [-18.981, -45.858, 111.161, 128.32, 74.084, 109.136, -572.14]
  MoveL 392 to (-72.16, 222.75, 20) mm, rotated rx 180 ry 50 rz 117.3 deg; joints [-19.385, -45.888, 111.176, 127.919, 74.208, 109.256, -567.303]
  MoveL 393 to (-74.48, 228.68, 10) mm, rotated rx -180 ry 50 rz 112.81 deg; joints [-19.79, -45.914, 111.185, 127.519, 74.332, 109.378, -562.811]
  MoveL 394 to (-76.17, 234.21, 0) mm, rotated rx 180 ry 50 rz 108.7 deg; joints [-20.194, -45.935, 111.187, 127.118, 74.455, 109.5, -558.703]
  MoveL 395 to (78.63, 249.2, 290) mm, rotated rx 180 ry 50 rz -97.82 deg; joints [-8.613, -44.864, 108.67, 138.329, 69.824, 107.066, -712.181]
  Set speed (60.0 mm/s)
  MoveL 396 to (58.93, 255.88, 290) mm, rotated rx 180 ry 50 rz -94 deg; joints [-8.613, -45.973, 108.773, 138.077, 69.074, 107.782, -715.998]
  MoveL 397 to (-76.17, 234.21, 0) mm, rotated rx -180 ry 50 rz 108.7 deg; joints [-20.194, -45.935, 111.187, 127.118, 74.455, 109.5, -558.703]
  Set speed (60.0 mm/s)
  MoveL 398 to (-55.37, 234.2, 0) mm, rotated rx 180 ry 50 rz 114.99 deg; joints [-20.194, -47.02, 111.288, 126.896, 73.863, 110.316, -564.986]
  MoveL 399 to (-76.17, 234.21, 0) mm, rotated rx -180 ry 50 rz 108.7 deg; joints [-20.194, -45.935, 111.187, 127.118, 74.455, 109.5, -558.703]
  Set speed (60.0 mm/s)
  MoveL 400 to (-74.48, 228.68, 10) mm, rotated rx -180 ry 50 rz 112.81 deg; joints [-19.79, -45.914, 111.185, 127.519, 74.332, 109.378, -562.811]
  MoveL 401 to (-72.16, 222.75, 20) mm, rotated rx 180 ry 50 rz 117.3 deg; joints [-19.385, -45.888, 111.176, 127.919, 74.208, 109.256, -567.303]
  MoveL 402 to (-69.12, 216.58, 30) mm, rotated rx 180 ry 50 rz 122.14 deg; joints [-18.981, -45.858, 111.161, 128.32, 74.084, 109.136, -572.14]
  MoveL 403 to (-65.29, 210.3, 40) mm, rotated rx 180 ry 50 rz 127.28 deg; joints [-18.576, -45.826, 111.139, 128.72, 73.959, 109.018, -577.284]
  MoveL 404 to (-60.61, 204.07, 50) mm, rotated rx -180 ry 50 rz 132.7 deg; joints [-18.172, -45.791, 111.112, 129.119, 73.832, 108.901, -582.698]
  MoveL 405 to (-55.08, 198.08, 60) mm, rotated rx 180 ry 50 rz 138.35 deg; joints [-17.768, -45.754, 111.078, 129.518, 73.703, 108.788, -588.347]
  MoveL 406 to (-48.7, 192.48, 70) mm, rotated rx -180 ry 50 rz 144.2 deg; joints [-17.364, -45.717, 111.038, 129.916, 73.572, 108.677, -594.197]
  MoveL 407 to (-41.52, 187.45, 80) mm, rotated rx 180 ry 50 rz 150.21 deg; joints [-16.96, -45.678, 110.993, 130.314, 73.439, 108.57, -600.214]
  MoveL 408 to (-33.62, 183.16, 90) mm, rotated rx -180 ry 50 rz 156.37 deg; joints [-16.557, -45.64, 110.941, 130.71, 73.302, 108.466, -606.369]
  MoveL 409 to (-25.11, 179.73, 100) mm, rotated rx -180 ry 50 rz 162.63 deg; joints [-16.154, -45.602, 110.884, 131.105, 73.162, 108.366, -612.629]
  MoveL 410 to (-16.13, 177.3, 110) mm, rotated rx -180 ry 50 rz 168.97 deg; joints [-15.751, -45.566, 110.82, 131.498, 73.018, 108.271, -618.967]
  MoveL 411 to (-6.83, 175.92, 120) mm, rotated rx -180 ry 50 rz 175.35 deg; joints [-15.349, -45.53, 110.751, 131.89, 72.869, 108.18, -625.352]
  MoveL 412 to (2.59, 175.67, 130) mm, rotated rx -180 ry 50 rz -178.24 deg; joints [-14.948, -45.496, 110.677, 132.28, 72.717, 108.093, -631.758]
  MoveL 413 to (11.96, 176.54, 140) mm, rotated rx -180 ry 50 rz -171.84 deg; joints [-14.546, -45.464, 110.596, 132.669, 72.561, 108.011, -638.157]
  MoveL 414 to (21.11, 178.51, 150) mm, rotated rx -180 ry 50 rz -165.48 deg; joints [-14.146, -45.432, 110.51, 133.056, 72.4, 107.933, -644.519]
  MoveL 415 to (29.85, 181.5, 160) mm, rotated rx -180 ry 50 rz -159.18 deg; joints [-13.746, -45.402, 110.418, 133.441, 72.234, 107.859, -650.818]
  MoveL 416 to (38.04, 185.42, 170) mm, rotated rx 180 ry 50 rz -152.98 deg; joints [-13.346, -45.372, 110.32, 133.825, 72.065, 107.788, -657.024]
  MoveL 417 to (45.56, 190.13, 180) mm, rotated rx 180 ry 50 rz -146.89 deg; joints [-12.947, -45.343, 110.216, 134.207, 71.892, 107.721, -663.107]
  MoveL 418 to (52.31, 195.49, 190) mm, rotated rx 180 ry 50 rz -140.96 deg; joints [-12.549, -45.313, 110.107, 134.587, 71.715, 107.656, -669.037]
  MoveL 419 to (58.22, 201.33, 200) mm, rotated rx -180 ry 50 rz -135.22 deg; joints [-12.152, -45.282, 109.991, 134.966, 71.535, 107.594, -674.781]
  MoveL 420 to (63.28, 207.47, 210) mm, rotated rx -180 ry 50 rz -129.69 deg; joints [-11.755, -45.25, 109.87, 135.344, 71.352, 107.533, -680.305]
  MoveL 421 to (67.49, 213.75, 220) mm, rotated rx 180 ry 50 rz -124.42 deg; joints [-11.359, -45.216, 109.742, 135.721, 71.166, 107.474, -685.575]
  MoveL 422 to (70.88, 219.99, 230) mm, rotated rx 180 ry 50 rz -119.44 deg; joints [-10.964, -45.178, 109.608, 136.096, 70.978, 107.416, -690.555]
  MoveL 423 to (73.51, 226.04, 240) mm, rotated rx 180 ry 50 rz -114.79 deg; joints [-10.57, -45.137, 109.467, 136.47, 70.789, 107.358, -695.208]
  MoveL 424 to (75.48, 231.77, 250) mm, rotated rx 180 ry 50 rz -110.51 deg; joints [-10.177, -45.092, 109.321, 136.844, 70.597, 107.301, -699.493]
  MoveL 425 to (76.86, 237.05, 260) mm, rotated rx -180 ry 50 rz -106.63 deg; joints [-9.784, -45.043, 109.168, 137.216, 70.405, 107.243, -703.374]
  MoveL 426 to (77.78, 241.77, 270) mm, rotated rx 180 ry 50 rz -103.19 deg; joints [-9.393, -44.989, 109.008, 137.588, 70.212, 107.185, -706.809]
  MoveL 427 to (78.34, 245.85, 280) mm, rotated rx -180 ry 50 rz -100.24 deg; joints [-9.003, -44.929, 108.842, 137.958, 70.018, 107.126, -709.758]
  MoveL 428 to (78.63, 249.2, 290) mm, rotated rx 180 ry 50 rz -97.82 deg; joints [-8.613, -44.864, 108.67, 138.329, 69.824, 107.066, -712.181]
  MoveL 429 to (58.93, 255.88, 290) mm, rotated rx 180 ry 50 rz -94 deg; joints [-8.613, -45.973, 108.773, 138.077, 69.074, 107.782, -715.998]
  Set speed (60.0 mm/s)
  MoveL 430 to (58.94, 253.36, 280) mm, rotated rx 180 ry 50 rz -96.43 deg; joints [-9.003, -46.04, 108.946, 137.708, 69.271, 107.848, -713.568]
  MoveL 431 to (58.8, 250.28, 270) mm, rotated rx 180 ry 50 rz -99.38 deg; joints [-9.393, -46.102, 109.112, 137.337, 69.468, 107.912, -710.615]
  MoveL 432 to (58.44, 246.7, 260) mm, rotated rx 180 ry 50 rz -102.82 deg; joints [-9.784, -46.158, 109.272, 136.966, 69.665, 107.975, -707.181]
  MoveL 433 to (57.77, 242.68, 250) mm, rotated rx 180 ry 50 rz -106.69 deg; joints [-10.177, -46.209, 109.426, 136.594, 69.861, 108.037, -703.306]
  MoveL 434 to (56.69, 238.28, 240) mm, rotated rx 180 ry 50 rz -110.97 deg; joints [-10.57, -46.255, 109.573, 136.222, 70.057, 108.1, -699.034]
  MoveL 435 to (55.14, 233.59, 230) mm, rotated rx 180 ry 50 rz -115.59 deg; joints [-10.964, -46.297, 109.714, 135.848, 70.251, 108.162, -694.405]
  MoveL 436 to (53.04, 228.71, 220) mm, rotated rx -180 ry 50 rz -120.54 deg; joints [-11.359, -46.335, 109.849, 135.474, 70.443, 108.224, -689.46]
  MoveL 437 to (50.33, 223.75, 210) mm, rotated rx -180 ry 50 rz -125.76 deg; joints [-11.755, -46.37, 109.977, 135.098, 70.633, 108.287, -684.235]
  MoveL 438 to (46.98, 218.83, 200) mm, rotated rx 180 ry 50 rz -131.23 deg; joints [-12.152, -46.403, 110.1, 134.722, 70.821, 108.352, -678.769]
  MoveL 439 to (42.97, 214.08, 190) mm, rotated rx 180 ry 50 rz -136.9 deg; joints [-12.549, -46.433, 110.216, 134.344, 71.007, 108.418, -673.096]
  MoveL 440 to (38.31, 209.62, 180) mm, rotated rx 180 ry 50 rz -142.75 deg; joints [-12.947, -46.463, 110.326, 133.964, 71.189, 108.486, -667.251]
  MoveL 441 to (33.03, 205.6, 170) mm, rotated rx 180 ry 50 rz -148.74 deg; joints [-13.346, -46.492, 110.43, 133.584, 71.368, 108.557, -661.263]
  MoveL 442 to (27.19, 202.13, 160) mm, rotated rx -180 ry 50 rz -154.84 deg; joints [-13.746, -46.52, 110.528, 133.201, 71.543, 108.63, -655.164]
  MoveL 443 to (20.88, 199.3, 150) mm, rotated rx 180 ry 50 rz -161.02 deg; joints [-14.146, -46.549, 110.62, 132.817, 71.714, 108.708, -648.983]
  MoveL 444 to (14.2, 197.22, 140) mm, rotated rx -180 ry 50 rz -167.25 deg; joints [-14.546, -46.579, 110.706, 132.431, 71.881, 108.788, -642.746]
  MoveL 445 to (7.28, 195.93, 130) mm, rotated rx -180 ry 50 rz -173.52 deg; joints [-14.948, -46.609, 110.787, 132.044, 72.044, 108.873, -636.481]
  MoveL 446 to (0.24, 195.48, 120) mm, rotated rx 180 ry 50 rz -179.79 deg; joints [-15.349, -46.641, 110.861, 131.655, 72.203, 108.963, -630.213]
  MoveL 447 to (-6.77, 195.87, 110) mm, rotated rx 180 ry 50 rz 173.97 deg; joints [-15.751, -46.674, 110.93, 131.264, 72.357, 109.056, -623.969]
  MoveL 448 to (-13.63, 197.08, 100) mm, rotated rx 180 ry 50 rz 167.78 deg; joints [-16.154, -46.708, 110.993, 130.872, 72.508, 109.154, -617.775]
  MoveL 449 to (-20.21, 199.05, 90) mm, rotated rx 180 ry 50 rz 161.66 deg; joints [-16.557, -46.743, 111.049, 130.478, 72.655, 109.256, -611.658]
  MoveL 450 to (-26.38, 201.72, 80) mm, rotated rx 180 ry 50 rz 155.64 deg; joints [-16.96, -46.779, 111.1, 130.084, 72.798, 109.362, -605.644]
  MoveL 451 to (-32.08, 204.97, 70) mm, rotated rx 180 ry 50 rz 149.76 deg; joints [-17.364, -46.814, 111.145, 129.687, 72.938, 109.472, -599.763]
  MoveL 452 to (-37.21, 208.71, 60) mm, rotated rx -180 ry 50 rz 144.04 deg; joints [-17.768, -46.85, 111.184, 129.29, 73.075, 109.585, -594.043]
  MoveL 453 to (-41.73, 212.8, 50) mm, rotated rx 180 ry 50 rz 138.52 deg; joints [-18.172, -46.884, 111.217, 128.892, 73.21, 109.702, -588.517]
  MoveL 454 to (-45.64, 217.12, 40) mm, rotated rx 180 ry 50 rz 133.22 deg; joints [-18.576, -46.917, 111.244, 128.494, 73.343, 109.821, -583.217]
  MoveL 455 to (-48.92, 221.54, 30) mm, rotated rx 180 ry 50 rz 128.18 deg; joints [-18.981, -46.947, 111.264, 128.094, 73.475, 109.943, -578.176]
  MoveL 456 to (-51.6, 225.93, 20) mm, rotated rx -180 ry 50 rz 123.43 deg; joints [-19.385, -46.975, 111.279, 127.695, 73.605, 110.066, -573.433]
  MoveL 457 to (-53.73, 230.19, 10) mm, rotated rx -180 ry 50 rz 119.02 deg; joints [-19.79, -46.999, 111.287, 127.295, 73.734, 110.191, -569.023]
  MoveL 458 to (-55.37, 234.2, 0) mm, rotated rx -180 ry 50 rz 114.99 deg; joints [-20.194, -47.02, 111.288, 126.896, 73.863, 110.316, -564.986]
  MoveL 459 to (58.93, 255.88, 290) mm, rotated rx 180 ry 50 rz -94 deg; joints [-8.613, -45.973, 108.773, 138.077, 69.074, 107.782, -715.998]
  Set speed (60.0 mm/s)
  MoveL 460 to (37.11, 300.24, 290) mm, rotated rx 180 ry 50 rz -42.69 deg; joints [-8.613, -46.208, 108.79, 138.021, 68.912, 107.938, -767.315]
  MoveL 461 to (-55.37, 234.2, 0) mm, rotated rx -180 ry 50 rz 114.99 deg; joints [-20.194, -47.02, 111.288, 126.896, 73.863, 110.316, -924.986]
  Set speed (60.0 mm/s)
  MoveL 462 to (-20.49, 199.16, 0) mm, rotated rx -180 ry 50 rz 161.39 deg; joints [-20.194, -46.846, 111.274, 126.932, 73.959, 110.184, -971.385]
  MoveL 463 to (-55.37, 234.2, 0) mm, rotated rx 180 ry 50 rz 114.99 deg; joints [-20.194, -47.02, 111.288, 126.896, 73.863, 110.316, -924.986]
  Set speed (60.0 mm/s)
  MoveL 464 to (-53.73, 230.19, 10) mm, rotated rx -180 ry 50 rz 119.02 deg; joints [-19.79, -46.999, 111.287, 127.295, 73.734, 110.191, -929.023]
  MoveL 465 to (-51.6, 225.93, 20) mm, rotated rx 180 ry 50 rz 123.43 deg; joints [-19.385, -46.975, 111.279, 127.695, 73.605, 110.066, -933.433]
  MoveL 466 to (-48.92, 221.54, 30) mm, rotated rx -180 ry 50 rz 128.18 deg; joints [-18.981, -46.947, 111.264, 128.094, 73.475, 109.943, -938.176]
  MoveL 467 to (-45.64, 217.12, 40) mm, rotated rx 180 ry 50 rz 133.22 deg; joints [-18.576, -46.917, 111.244, 128.494, 73.343, 109.821, -943.217]
  MoveL 468 to (-41.73, 212.8, 50) mm, rotated rx 180 ry 50 rz 138.52 deg; joints [-18.172, -46.884, 111.217, 128.892, 73.21, 109.702, -948.517]
  MoveL 469 to (-37.21, 208.71, 60) mm, rotated rx 180 ry 50 rz 144.04 deg; joints [-17.768, -46.85, 111.184, 129.29, 73.075, 109.585, -954.043]
  MoveL 470 to (-32.08, 204.97, 70) mm, rotated rx -180 ry 50 rz 149.76 deg; joints [-17.364, -46.814, 111.145, 129.687, 72.938, 109.472, -959.763]
  MoveL 471 to (-26.38, 201.72, 80) mm, rotated rx 180 ry 50 rz 155.64 deg; joints [-16.96, -46.779, 111.1, 130.084, 72.798, 109.362, -965.644]
  MoveL 472 to (-20.21, 199.05, 90) mm, rotated rx -180 ry 50 rz 161.66 deg; joints [-16.557, -46.743, 111.049, 130.478, 72.655, 109.256, -971.658]
  MoveL 473 to (-13.63, 197.08, 100) mm, rotated rx 180 ry 50 rz 167.78 deg; joints [-16.154, -46.708, 110.993, 130.872, 72.508, 109.154, -977.775]
  MoveL 474 to (-6.77, 195.87, 110) mm, rotated rx 180 ry 50 rz 173.97 deg; joints [-15.751, -46.674, 110.93, 131.264, 72.357, 109.056, -983.969]
  MoveL 475 to (0.24, 195.48, 120) mm, rotated rx 180 ry 50 rz -179.79 deg; joints [-15.349, -46.641, 110.861, 131.655, 72.203, 108.963, -990.213]
  MoveL 476 to (7.28, 195.93, 130) mm, rotated rx 180 ry 50 rz -173.52 deg; joints [-14.948, -46.609, 110.787, 132.044, 72.044, 108.873, -996.481]
  MoveL 477 to (14.2, 197.22, 140) mm, rotated rx -180 ry 50 rz -167.25 deg; joints [-14.546, -46.579, 110.706, 132.431, 71.881, 108.788, -1002.746]
  MoveL 478 to (20.88, 199.3, 150) mm, rotated rx -180 ry 50 rz -161.02 deg; joints [-14.146, -46.549, 110.62, 132.817, 71.714, 108.708, -1008.983]
  MoveL 479 to (27.19, 202.13, 160) mm, rotated rx -180 ry 50 rz -154.84 deg; joints [-13.746, -46.52, 110.528, 133.201, 71.543, 108.63, -1015.164]
  MoveL 480 to (33.03, 205.6, 170) mm, rotated rx -180 ry 50 rz -148.74 deg; joints [-13.346, -46.492, 110.43, 133.584, 71.368, 108.557, -1021.263]
  MoveL 481 to (38.31, 209.62, 180) mm, rotated rx 180 ry 50 rz -142.75 deg; joints [-12.947, -46.463, 110.326, 133.964, 71.189, 108.486, -1027.251]
  MoveL 482 to (42.97, 214.08, 190) mm, rotated rx -180 ry 50 rz -136.9 deg; joints [-12.549, -46.433, 110.216, 134.344, 71.007, 108.418, -1033.096]
  MoveL 483 to (46.98, 218.83, 200) mm, rotated rx 180 ry 50 rz -131.23 deg; joints [-12.152, -46.403, 110.1, 134.722, 70.821, 108.352, -1038.769]
  MoveL 484 to (50.33, 223.75, 210) mm, rotated rx -180 ry 50 rz -125.76 deg; joints [-11.755, -46.37, 109.977, 135.098, 70.633, 108.287, -1044.235]
  MoveL 485 to (53.04, 228.71, 220) mm, rotated rx -180 ry 50 rz -120.54 deg; joints [-11.359, -46.335, 109.849, 135.474, 70.443, 108.224, -1049.46]
  MoveL 486 to (55.14, 233.59, 230) mm, rotated rx -180 ry 50 rz -115.59 deg; joints [-10.964, -46.297, 109.714, 135.848, 70.251, 108.162, -1054.405]
  MoveL 487 to (56.69, 238.28, 240) mm, rotated rx 180 ry 50 rz -110.97 deg; joints [-10.57, -46.255, 109.573, 136.222, 70.057, 108.1, -1059.034]
  MoveL 488 to (57.77, 242.68, 250) mm, rotated rx -180 ry 50 rz -106.69 deg; joints [-10.177, -46.209, 109.426, 136.594, 69.861, 108.037, -1063.306]
  MoveL 489 to (58.44, 246.7, 260) mm, rotated rx -180 ry 50 rz -102.82 deg; joints [-9.784, -46.158, 109.272, 136.966, 69.665, 107.975, -1067.181]
  MoveL 490 to (58.8, 250.28, 270) mm, rotated rx 180 ry 50 rz -99.38 deg; joints [-9.393, -46.102, 109.112, 137.337, 69.468, 107.912, -1070.615]
  MoveL 491 to (58.94, 253.36, 280) mm, rotated rx -180 ry 50 rz -96.43 deg; joints [-9.003, -46.04, 108.946, 137.708, 69.271, 107.848, -1073.568]
  MoveL 492 to (58.93, 255.88, 290) mm, rotated rx 180 ry 50 rz -94 deg; joints [-8.613, -45.973, 108.773, 138.077, 69.074, 107.782, -1075.998]
  MoveL 493 to (37.11, 300.24, 290) mm, rotated rx 180 ry 50 rz -42.69 deg; joints [-8.613, -46.208, 108.79, 138.021, 68.912, 107.938, -1127.315]
  Set speed (60.0 mm/s)
  MoveL 494 to (39.03, 298.61, 280) mm, rotated rx 180 ry 50 rz -45.31 deg; joints [-9.003, -46.28, 108.964, 137.651, 69.107, 108.007, -1124.686]
  MoveL 495 to (41.29, 296.51, 270) mm, rotated rx 180 ry 50 rz -48.51 deg; joints [-9.393, -46.346, 109.131, 137.28, 69.303, 108.075, -1121.487]
  MoveL 496 to (43.78, 293.91, 260) mm, rotated rx -180 ry 50 rz -52.23 deg; joints [-9.784, -46.406, 109.291, 136.908, 69.497, 108.142, -1117.765]
  MoveL 497 to (46.4, 290.79, 250) mm, rotated rx 180 ry 50 rz -56.43 deg; joints [-10.177, -46.461, 109.445, 136.535, 69.692, 108.208, -1113.565]
  MoveL 498 to (49.06, 287.12, 240) mm, rotated rx 180 ry 50 rz -61.06 deg; joints [-10.57, -46.51, 109.593, 136.163, 69.887, 108.273, -1108.935]
  MoveL 499 to (51.62, 282.9, 230) mm, rotated rx 180 ry 50 rz -66.08 deg; joints [-10.964, -46.553, 109.734, 135.789, 70.081, 108.337, -1103.922]
  MoveL 500 to (53.98, 278.14, 220) mm, rotated rx 180 ry 50 rz -71.43 deg; joints [-11.359, -46.59, 109.869, 135.415, 70.275, 108.399, -1098.571]
  MoveL 501 to (56, 272.86, 210) mm, rotated rx 180 ry 50 rz -77.07 deg; joints [-11.755, -46.622, 109.997, 135.041, 70.469, 108.461, -1092.931]
  MoveL 502 to (57.57, 267.12, 200) mm, rotated rx 180 ry 50 rz -82.95 deg; joints [-12.152, -46.649, 110.119, 134.666, 70.662, 108.522, -1087.046]
  MoveL 503 to (58.59, 260.98, 190) mm, rotated rx -180 ry 50 rz -89.04 deg; joints [-12.549, -46.671, 110.235, 134.29, 70.854, 108.583, -1080.96]
  MoveL 504 to (58.95, 254.55, 180) mm, rotated rx -180 ry 50 rz -95.29 deg; joints [-12.947, -46.688, 110.344, 133.913, 71.045, 108.644, -1074.714]
  MoveL 505 to (58.59, 247.92, 170) mm, rotated rx 180 ry 50 rz -101.65 deg; joints [-13.346, -46.703, 110.447, 133.536, 71.234, 108.705, -1068.348]
  MoveL 506 to (57.45, 241.22, 160) mm, rotated rx 180 ry 50 rz -108.1 deg; joints [-13.746, -46.714, 110.544, 133.158, 71.421, 108.767, -1061.898]
  MoveL 507 to (55.51, 234.59, 150) mm, rotated rx 180 ry 50 rz -114.6 deg; joints [-14.146, -46.723, 110.634, 132.778, 71.606, 108.831, -1055.4]
  MoveL 508 to (52.77, 228.15, 140) mm, rotated rx -180 ry 50 rz -121.12 deg; joints [-14.546, -46.73, 110.719, 132.398, 71.787, 108.897, -1048.885]
  MoveL 509 to (49.26, 222.05, 130) mm, rotated rx 180 ry 50 rz -127.62 deg; joints [-14.948, -46.737, 110.797, 132.016, 71.966, 108.965, -1042.384]
  MoveL 510 to (45.04, 216.4, 120) mm, rotated rx 180 ry 50 rz -134.07 deg; joints [-15.349, -46.743, 110.87, 131.633, 72.141, 109.036, -1035.926]
  MoveL 511 to (40.19, 211.31, 110) mm, rotated rx 180 ry 50 rz -140.46 deg; joints [-15.751, -46.749, 110.936, 131.248, 72.312, 109.11, -1029.537]
  MoveL 512 to (34.83, 206.87, 100) mm, rotated rx -180 ry 50 rz -146.76 deg; joints [-16.154, -46.756, 110.997, 130.862, 72.479, 109.188, -1023.245]
  MoveL 513 to (29.06, 203.14, 90) mm, rotated rx -180 ry 50 rz -152.93 deg; joints [-16.557, -46.763, 111.051, 130.474, 72.643, 109.27, -1017.074]
  MoveL 514 to (23.03, 200.17, 80) mm, rotated rx -180 ry 50 rz -158.95 deg; joints [-16.96, -46.771, 111.1, 130.085, 72.802, 109.357, -1011.051]
  MoveL 515 to (16.86, 197.94, 70) mm, rotated rx -180 ry 50 rz -164.8 deg; joints [-17.364, -46.78, 111.142, 129.695, 72.958, 109.447, -1005.201]
  MoveL 516 to (10.69, 196.46, 60) mm, rotated rx 180 ry 50 rz -170.45 deg; joints [-17.768, -46.79, 111.179, 129.303, 73.11, 109.541, -999.549]
  MoveL 517 to (4.64, 195.67, 50) mm, rotated rx -180 ry 50 rz -175.88 deg; joints [-18.172, -46.8, 111.21, 128.91, 73.258, 109.64, -994.124]
  MoveL 518 to (-1.18, 195.49, 40) mm, rotated rx -180 ry 50 rz 178.95 deg; joints [-18.576, -46.811, 111.235, 128.516, 73.404, 109.742, -988.952]
  MoveL 519 to (-6.67, 195.86, 30) mm, rotated rx -180 ry 50 rz 174.06 deg; joints [-18.981, -46.821, 111.254, 128.121, 73.546, 109.848, -984.062]
  MoveL 520 to (-11.76, 196.67, 20) mm, rotated rx -180 ry 50 rz 169.48 deg; joints [-19.385, -46.831, 111.267, 127.726, 73.686, 109.957, -979.483]
  MoveL 521 to (-16.38, 197.8, 10) mm, rotated rx 180 ry 50 rz 165.25 deg; joints [-19.79, -46.839, 111.274, 127.329, 73.823, 110.069, -975.247]
  MoveL 522 to (-20.49, 199.16, 0) mm, rotated rx 180 ry 50 rz 161.39 deg; joints [-20.194, -46.846, 111.274, 126.932, 73.959, 110.184, -971.385]
  MoveL 523 to (37.11, 300.24, 290) mm, rotated rx -180 ry 50 rz -42.69 deg; joints [-8.613, -46.208, 108.79, 138.021, 68.912, 107.938, -1127.315]
  Set speed (60.0 mm/s)
  MoveL 524 to (43.85, 319.91, 290) mm, rotated rx -180 ry 50 rz -36.2 deg; joints [-8.613, -45.145, 108.699, 138.267, 69.635, 107.245, -1133.803]
  MoveL 525 to (-20.49, 199.16, 0) mm, rotated rx 180 ry 50 rz 161.39 deg; joints [-20.194, -46.846, 111.274, 126.932, 73.959, 110.184, -971.385]
  Set speed (60.0 mm/s)
  MoveL 526 to (-20.57, 178.36, 0) mm, rotated rx -180 ry 50 rz 165.86 deg; joints [-20.194, -45.722, 111.164, 127.16, 74.569, 109.343, -975.856]
  MoveL 527 to (-20.49, 199.16, 0) mm, rotated rx 180 ry 50 rz 161.39 deg; joints [-20.194, -46.846, 111.274, 126.932, 73.959, 110.184, -971.385]
  Set speed (60.0 mm/s)
  MoveL 528 to (-16.38, 197.8, 10) mm, rotated rx 180 ry 50 rz 165.25 deg; joints [-19.79, -46.839, 111.274, 127.329, 73.823, 110.069, -975.247]
  MoveL 529 to (-11.76, 196.67, 20) mm, rotated rx 180 ry 50 rz 169.48 deg; joints [-19.385, -46.831, 111.267, 127.726, 73.686, 109.957, -979.483]
  MoveL 530 to (-6.67, 195.86, 30) mm, rotated rx -180 ry 50 rz 174.06 deg; joints [-18.981, -46.821, 111.254, 128.121, 73.546, 109.848, -984.062]
  MoveL 531 to (-1.18, 195.49, 40) mm, rotated rx 180 ry 50 rz 178.95 deg; joints [-18.576, -46.811, 111.235, 128.516, 73.404, 109.742, -988.952]
  MoveL 532 to (4.64, 195.67, 50) mm, rotated rx -180 ry 50 rz -175.88 deg; joints [-18.172, -46.8, 111.21, 128.91, 73.258, 109.64, -994.124]
  MoveL 533 to (10.69, 196.46, 60) mm, rotated rx -180 ry 50 rz -170.45 deg; joints [-17.768, -46.79, 111.179, 129.303, 73.11, 109.541, -999.549]
  MoveL 534 to (16.86, 197.94, 70) mm, rotated rx 180 ry 50 rz -164.8 deg; joints [-17.364, -46.78, 111.142, 129.695, 72.958, 109.447, -1005.201]
  MoveL 535 to (23.03, 200.17, 80) mm, rotated rx 180 ry 50 rz -158.95 deg; joints [-16.96, -46.771, 111.1, 130.085, 72.802, 109.357, -1011.051]
  MoveL 536 to (29.06, 203.14, 90) mm, rotated rx 180 ry 50 rz -152.93 deg; joints [-16.557, -46.763, 111.051, 130.474, 72.643, 109.27, -1017.074]
  MoveL 537 to (34.83, 206.87, 100) mm, rotated rx 180 ry 50 rz -146.76 deg; joints [-16.154, -46.756, 110.997, 130.862, 72.479, 109.188, -1023.245]
  MoveL 538 to (40.19, 211.31, 110) mm, rotated rx -180 ry 50 rz -140.46 deg; joints [-15.751, -46.749, 110.936, 131.248, 72.312, 109.11, -1029.537]
  MoveL 539 to (45.04, 216.4, 120) mm, rotated rx 180 ry 50 rz -134.07 deg; joints [-15.349, -46.743, 110.87, 131.633, 72.141, 109.036, -1035.926]
  MoveL 540 to (49.26, 222.05, 130) mm, rotated rx -180 ry 50 rz -127.62 deg; joints [-14.948, -46.737, 110.797, 132.016, 71.966, 108.965, -1042.384]
  MoveL 541 to (52.77, 228.15, 140) mm, rotated rx 180 ry 50 rz -121.12 deg; joints [-14.546, -46.73, 110.719, 132.398, 71.787, 108.897, -1048.885]
  MoveL 542 to (55.51, 234.59, 150) mm, rotated rx -180 ry 50 rz -114.6 deg; joints [-14.146, -46.723, 110.634, 132.778, 71.606, 108.831, -1055.4]
  MoveL 543 to (57.45, 241.22, 160) mm, rotated rx -180 ry 50 rz -108.1 deg; joints [-13.746, -46.714, 110.544, 133.158, 71.421, 108.767, -1061.898]
  MoveL 544 to (58.59, 247.92, 170) mm, rotated rx 180 ry 50 rz -101.65 deg; joints [-13.346, -46.703, 110.447, 133.536, 71.234, 108.705, -1068.348]
  MoveL 545 to (58.95, 254.55, 180) mm, rotated rx 180 ry 50 rz -95.29 deg; joints [-12.947, -46.688, 110.344, 133.913, 71.045, 108.644, -1074.714]
  MoveL 546 to (58.59, 260.98, 190) mm, rotated rx 180 ry 50 rz -89.04 deg; joints [-12.549, -46.671, 110.235, 134.29, 70.854, 108.583, -1080.96]
  MoveL 547 to (57.57, 267.12, 200) mm, rotated rx -180 ry 50 rz -82.95 deg; joints [-12.152, -46.649, 110.119, 134.666, 70.662, 108.522, -1087.046]
  MoveL 548 to (56, 272.86, 210) mm, rotated rx 180 ry 50 rz -77.07 deg; joints [-11.755, -46.622, 109.997, 135.041, 70.469, 108.461, -1092.931]
  MoveL 549 to (53.98, 278.14, 220) mm, rotated rx 180 ry 50 rz -71.43 deg; joints [-11.359, -46.59, 109.869, 135.415, 70.275, 108.399, -1098.571]
  MoveL 550 to (51.62, 282.9, 230) mm, rotated rx 180 ry 50 rz -66.08 deg; joints [-10.964, -46.553, 109.734, 135.789, 70.081, 108.337, -1103.922]
  MoveL 551 to (49.06, 287.12, 240) mm, rotated rx 180 ry 50 rz -61.06 deg; joints [-10.57, -46.51, 109.593, 136.163, 69.887, 108.273, -1108.935]
  MoveL 552 to (46.4, 290.79, 250) mm, rotated rx 180 ry 50 rz -56.43 deg; joints [-10.177, -46.461, 109.445, 136.535, 69.692, 108.208, -1113.565]
  MoveL 553 to (43.78, 293.91, 260) mm, rotated rx 180 ry 50 rz -52.23 deg; joints [-9.784, -46.406, 109.291, 136.908, 69.497, 108.142, -1117.765]
  MoveL 554 to (41.29, 296.51, 270) mm, rotated rx -180 ry 50 rz -48.51 deg; joints [-9.393, -46.346, 109.131, 137.28, 69.303, 108.075, -1121.487]
  MoveL 555 to (39.03, 298.61, 280) mm, rotated rx -180 ry 50 rz -45.31 deg; joints [-9.003, -46.28, 108.964, 137.651, 69.107, 108.007, -1124.686]
  MoveL 556 to (37.11, 300.24, 290) mm, rotated rx 180 ry 50 rz -42.69 deg; joints [-8.613, -46.208, 108.79, 138.021, 68.912, 107.938, -1127.315]
  MoveL 557 to (43.85, 319.91, 290) mm, rotated rx -180 ry 50 rz -36.2 deg; joints [-8.613, -45.145, 108.699, 138.267, 69.635, 107.245, -1133.803]
  Set speed (60.0 mm/s)
  MoveL 558 to (46.6, 317.98, 280) mm, rotated rx 180 ry 50 rz -38.79 deg; joints [-9.003, -45.216, 108.872, 137.895, 69.827, 107.31, -1131.207]
  MoveL 559 to (49.86, 315.46, 270) mm, rotated rx 180 ry 50 rz -41.95 deg; joints [-9.393, -45.282, 109.039, 137.524, 70.018, 107.373, -1128.046]
  MoveL 560 to (53.49, 312.31, 260) mm, rotated rx -180 ry 50 rz -45.64 deg; joints [-9.784, -45.341, 109.199, 137.151, 70.209, 107.436, -1124.36]
  MoveL 561 to (57.36, 308.47, 250) mm, rotated rx 180 ry 50 rz -49.81 deg; joints [-10.177, -45.396, 109.352, 136.778, 70.399, 107.498, -1120.194]
  MoveL 562 to (61.34, 303.9, 240) mm, rotated rx -180 ry 50 rz -54.41 deg; joints [-10.57, -45.444, 109.5, 136.404, 70.59, 107.559, -1115.591]
  MoveL 563 to (65.27, 298.59, 230) mm, rotated rx 180 ry 50 rz -59.4 deg; joints [-10.964, -45.487, 109.64, 136.03, 70.779, 107.619, -1110.596]
  MoveL 564 to (68.98, 292.54, 220) mm, rotated rx 180 ry 50 rz -64.75 deg; joints [-11.359, -45.524, 109.774, 135.655, 70.969, 107.678, -1105.253]
  MoveL 565 to (72.31, 285.76, 210) mm, rotated rx -180 ry 50 rz -70.39 deg; joints [-11.755, -45.555, 109.902, 135.279, 71.158, 107.736, -1099.605]
  MoveL 566 to (75.1, 278.3, 200) mm, rotated rx 180 ry 50 rz -76.3 deg; joints [-12.152, -45.581, 110.023, 134.903, 71.347, 107.793, -1093.697]
  MoveL 567 to (77.2, 270.26, 190) mm, rotated rx -180 ry 50 rz -82.43 deg; joints [-12.549, -45.602, 110.138, 134.526, 71.534, 107.85, -1087.571]
  MoveL 568 to (78.47, 261.74, 180) mm, rotated rx 180 ry 50 rz -88.73 deg; joints [-12.947, -45.618, 110.246, 134.149, 71.721, 107.906, -1081.269]
  MoveL 569 to (78.79, 252.87, 170) mm, rotated rx 180 ry 50 rz -95.17 deg; joints [-13.346, -45.63, 110.348, 133.771, 71.906, 107.963, -1074.829]
  MoveL 570 to (78.09, 243.82, 160) mm, rotated rx 180 ry 50 rz -101.71 deg; joints [-13.746, -45.639, 110.444, 133.392, 72.089, 108.02, -1068.29]
  MoveL 571 to (76.31, 234.75, 150) mm, rotated rx -180 ry 50 rz -108.31 deg; joints [-14.146, -45.646, 110.533, 133.011, 72.27, 108.079, -1061.689]
  MoveL 572 to (73.44, 225.85, 140) mm, rotated rx -180 ry 50 rz -114.94 deg; joints [-14.546, -45.65, 110.617, 132.63, 72.448, 108.139, -1055.058]
  MoveL 573 to (69.5, 217.29, 130) mm, rotated rx -180 ry 50 rz -121.57 deg; joints [-14.948, -45.653, 110.694, 132.248, 72.623, 108.202, -1048.432]
  MoveL 574 to (64.57, 209.26, 120) mm, rotated rx 180 ry 50 rz -128.16 deg; joints [-15.349, -45.656, 110.765, 131.864, 72.795, 108.267, -1041.84]
  MoveL 575 to (58.74, 201.9, 110) mm, rotated rx 180 ry 50 rz -134.69 deg; joints [-15.751, -45.658, 110.831, 131.479, 72.963, 108.335, -1035.313]
  MoveL 576 to (52.14, 195.34, 100) mm, rotated rx 180 ry 50 rz -141.12 deg; joints [-16.154, -45.661, 110.89, 131.093, 73.127, 108.407, -1028.879]
  MoveL 577 to (44.91, 189.68, 90) mm, rotated rx 180 ry 50 rz -147.43 deg; joints [-16.557, -45.665, 110.944, 130.705, 73.288, 108.483, -1022.567]
  MoveL 578 to (37.24, 184.98, 80) mm, rotated rx 180 ry 50 rz -153.6 deg; joints [-16.96, -45.669, 110.992, 130.315, 73.444, 108.563, -1016.403]
  MoveL 579 to (29.3, 181.28, 70) mm, rotated rx 180 ry 50 rz -159.58 deg; joints [-17.364, -45.675, 111.034, 129.925, 73.596, 108.647, -1010.416]
  MoveL 580 to (21.27, 178.55, 60) mm, rotated rx -180 ry 50 rz -165.37 deg; joints [-17.768, -45.681, 111.07, 129.533, 73.745, 108.735, -1004.633]
  MoveL 581 to (13.31, 176.76, 50) mm, rotated rx -180 ry 50 rz -170.92 deg; joints [-18.172, -45.688, 111.1, 129.14, 73.89, 108.828, -999.083]
  MoveL 582 to (5.58, 175.83, 40) mm, rotated rx 180 ry 50 rz -176.21 deg; joints [-18.576, -45.696, 111.125, 128.746, 74.031, 108.924, -993.794]
  MoveL 583 to (-1.77, 175.65, 30) mm, rotated rx -180 ry 50 rz 178.8 deg; joints [-18.981, -45.703, 111.144, 128.35, 74.17, 109.024, -988.796]
  MoveL 584 to (-8.64, 176.1, 20) mm, rotated rx -180 ry 50 rz 174.12 deg; joints [-19.385, -45.711, 111.156, 127.954, 74.305, 109.127, -984.119]
  MoveL 585 to (-14.93, 177.06, 10) mm, rotated rx 180 ry 50 rz 169.79 deg; joints [-19.79, -45.717, 111.163, 127.558, 74.438, 109.234, -979.795]
  MoveL 586 to (-20.57, 178.36, 0) mm, rotated rx -180 ry 50 rz 165.86 deg; joints [-20.194, -45.722, 111.164, 127.16, 74.569, 109.343, -975.856]
  MoveL 587 to (43.85, 319.91, 290) mm, rotated rx -180 ry 50 rz -36.2 deg; joints [-8.613, -45.145, 108.699, 138.267, 69.635, 107.245, -1133.803]
  Set speed (60.0 mm/s)
  MoveL 588 to (28.22, 306.19, 290) mm, rotated rx 180 ry 50 rz -31.42 deg; joints [-8.613, -46.241, 108.793, 138.013, 68.889, 107.96, -1138.582]
  MoveL 589 to (-20.57, 178.36, 0) mm, rotated rx -180 ry 50 rz 165.86 deg; joints [-20.194, -45.722, 111.164, 127.16, 74.569, 109.343, -975.856]
  Set speed (60.0 mm/s)
  MoveL 590 to (-10.16, 196.36, 0) mm, rotated rx -180 ry 50 rz 170.93 deg; joints [-20.194, -46.832, 111.273, 126.935, 73.966, 110.173, -980.929]
  MoveL 591 to (-20.57, 178.36, 0) mm, rotated rx -180 ry 50 rz 165.86 deg; joints [-20.194, -45.722, 111.164, 127.16, 74.569, 109.343, -975.856]
  Set speed (60.0 mm/s)
  MoveL 592 to (-14.93, 177.06, 10) mm, rotated rx 180 ry 50 rz 169.79 deg; joints [-19.79, -45.717, 111.163, 127.558, 74.438, 109.234, -979.795]
  MoveL 593 to (-8.64, 176.1, 20) mm, rotated rx 180 ry 50 rz 174.12 deg; joints [-19.385, -45.711, 111.156, 127.954, 74.305, 109.127, -984.119]
  MoveL 594 to (-1.77, 175.65, 30) mm, rotated rx -180 ry 50 rz 178.8 deg; joints [-18.981, -45.703, 111.144, 128.35, 74.17, 109.024, -988.796]
  MoveL 595 to (5.58, 175.83, 40) mm, rotated rx 180 ry 50 rz -176.21 deg; joints [-18.576, -45.696, 111.125, 128.746, 74.031, 108.924, -993.794]
  MoveL 596 to (13.31, 176.76, 50) mm, rotated rx -180 ry 50 rz -170.92 deg; joints [-18.172, -45.688, 111.1, 129.14, 73.89, 108.828, -999.083]
  MoveL 597 to (21.27, 178.55, 60) mm, rotated rx 180 ry 50 rz -165.37 deg; joints [-17.768, -45.681, 111.07, 129.533, 73.745, 108.735, -1004.633]
  MoveL 598 to (29.3, 181.28, 70) mm, rotated rx 180 ry 50 rz -159.58 deg; joints [-17.364, -45.675, 111.034, 129.925, 73.596, 108.647, -1010.416]
  MoveL 599 to (37.24, 184.98, 80) mm, rotated rx 180 ry 50 rz -153.6 deg; joints [-16.96, -45.669, 110.992, 130.315, 73.444, 108.563, -1016.403]
  MoveL 600 to (44.91, 189.68, 90) mm, rotated rx 180 ry 50 rz -147.43 deg; joints [-16.557, -45.665, 110.944, 130.705, 73.288, 108.483, -1022.567]
  MoveL 601 to (52.14, 195.34, 100) mm, rotated rx 180 ry 50 rz -141.12 deg; joints [-16.154, -45.661, 110.89, 131.093, 73.127, 108.407, -1028.879]
  MoveL 602 to (58.74, 201.9, 110) mm, rotated rx -180 ry 50 rz -134.69 deg; joints [-15.751, -45.658, 110.831, 131.479, 72.963, 108.335, -1035.313]
  MoveL 603 to (64.57, 209.26, 120) mm, rotated rx 180 ry 50 rz -128.16 deg; joints [-15.349, -45.656, 110.765, 131.864, 72.795, 108.267, -1041.84]
  MoveL 604 to (69.5, 217.29, 130) mm, rotated rx 180 ry 50 rz -121.57 deg; joints [-14.948, -45.653, 110.694, 132.248, 72.623, 108.202, -1048.432]
  MoveL 605 to (73.44, 225.85, 140) mm, rotated rx -180 ry 50 rz -114.94 deg; joints [-14.546, -45.65, 110.617, 132.63, 72.448, 108.139, -1055.058]
  MoveL 606 to (76.31, 234.75, 150) mm, rotated rx -180 ry 50 rz -108.31 deg; joints [-14.146, -45.646, 110.533, 133.011, 72.27, 108.079, -1061.689]
  MoveL 607 to (78.09, 243.82, 160) mm, rotated rx -180 ry 50 rz -101.71 deg; joints [-13.746, -45.639, 110.444, 133.392, 72.089, 108.02, -1068.29]
  MoveL 608 to (78.79, 252.87, 170) mm, rotated rx -180 ry 50 rz -95.17 deg; joints [-13.346, -45.63, 110.348, 133.771, 71.906, 107.963, -1074.829]
  MoveL 609 to (78.47, 261.74, 180) mm, rotated rx -180 ry 50 rz -88.73 deg; joints [-12.947, -45.618, 110.246, 134.149, 71.721, 107.906, -1081.269]
  MoveL 610 to (77.2, 270.26, 190) mm, rotated rx -180 ry 50 rz -82.43 deg; joints [-12.549, -45.602, 110.138, 134.526, 71.534, 107.85, -1087.571]
  MoveL 611 to (75.1, 278.3, 200) mm, rotated rx -180 ry 50 rz -76.3 deg; joints [-12.152, -45.581, 110.023, 134.903, 71.347, 107.793, -1093.697]
  MoveL 612 to (72.31, 285.76, 210) mm, rotated rx 180 ry 50 rz -70.39 deg; joints [-11.755, -45.555, 109.902, 135.279, 71.158, 107.736, -1099.605]
  MoveL 613 to (68.98, 292.54, 220) mm, rotated rx 180 ry 50 rz -64.75 deg; joints [-11.359, -45.524, 109.774, 135.655, 70.969, 107.678, -1105.253]
  MoveL 614 to (65.27, 298.59, 230) mm, rotated rx -180 ry 50 rz -59.4 deg; joints [-10.964, -45.487, 109.64, 136.03, 70.779, 107.619, -1110.596]
  MoveL 615 to (61.34, 303.9, 240) mm, rotated rx 180 ry 50 rz -54.41 deg; joints [-10.57, -45.444, 109.5, 136.404, 70.59, 107.559, -1115.591]
  MoveL 616 to (57.36, 308.47, 250) mm, rotated rx -180 ry 50 rz -49.81 deg; joints [-10.177, -45.396, 109.352, 136.778, 70.399, 107.498, -1120.194]
  MoveL 617 to (53.49, 312.31, 260) mm, rotated rx -180 ry 50 rz -45.64 deg; joints [-9.784, -45.341, 109.199, 137.151, 70.209, 107.436, -1124.36]
  MoveL 618 to (49.86, 315.46, 270) mm, rotated rx 180 ry 50 rz -41.95 deg; joints [-9.393, -45.282, 109.039, 137.524, 70.018, 107.373, -1128.046]
  MoveL 619 to (46.6, 317.98, 280) mm, rotated rx 180 ry 50 rz -38.79 deg; joints [-9.003, -45.216, 108.872, 137.895, 69.827, 107.31, -1131.207]
  MoveL 620 to (43.85, 319.91, 290) mm, rotated rx 180 ry 50 rz -36.2 deg; joints [-8.613, -45.145, 108.699, 138.267, 69.635, 107.245, -1133.803]
  MoveL 621 to (28.22, 306.19, 290) mm, rotated rx 180 ry 50 rz -31.42 deg; joints [-8.613, -46.241, 108.793, 138.013, 68.889, 107.96, -1138.582]
  Set speed (60.0 mm/s)
  MoveL 622 to (30.4, 304.94, 280) mm, rotated rx 180 ry 50 rz -34.08 deg; joints [-9.003, -46.315, 108.966, 137.642, 69.083, 108.031, -1135.919]
  MoveL 623 to (33, 303.28, 270) mm, rotated rx 180 ry 50 rz -37.32 deg; joints [-9.393, -46.383, 109.133, 137.271, 69.277, 108.1, -1132.679]
  MoveL 624 to (35.92, 301.18, 260) mm, rotated rx 180 ry 50 rz -41.09 deg; joints [-9.784, -46.446, 109.294, 136.898, 69.47, 108.169, -1128.905]
  MoveL 625 to (39.07, 298.58, 250) mm, rotated rx 180 ry 50 rz -45.36 deg; joints [-10.177, -46.504, 109.448, 136.525, 69.663, 108.237, -1124.643]
  MoveL 626 to (42.34, 295.45, 240) mm, rotated rx 180 ry 50 rz -50.06 deg; joints [-10.57, -46.555, 109.596, 136.152, 69.856, 108.304, -1119.941]
  MoveL 627 to (45.62, 291.76, 230) mm, rotated rx 180 ry 50 rz -55.15 deg; joints [-10.964, -46.601, 109.737, 135.778, 70.049, 108.37, -1114.846]
  MoveL 628 to (48.8, 287.5, 220) mm, rotated rx 180 ry 50 rz -60.59 deg; joints [-11.359, -46.641, 109.872, 135.403, 70.242, 108.434, -1109.406]
  MoveL 629 to (51.74, 282.68, 210) mm, rotated rx 180 ry 50 rz -66.33 deg; joints [-11.755, -46.675, 110.001, 135.028, 70.435, 108.498, -1103.668]
  MoveL 630 to (54.33, 277.32, 200) mm, rotated rx 180 ry 50 rz -72.32 deg; joints [-12.152, -46.703, 110.123, 134.653, 70.627, 108.56, -1097.679]
  MoveL 631 to (56.44, 271.47, 190) mm, rotated rx -180 ry 50 rz -78.51 deg; joints [-12.549, -46.726, 110.239, 134.277, 70.818, 108.622, -1091.486]
  MoveL 632 to (57.96, 265.2, 180) mm, rotated rx 180 ry 50 rz -84.87 deg; joints [-12.947, -46.744, 110.348, 133.901, 71.009, 108.683, -1085.13]
  MoveL 633 to (58.8, 258.62, 170) mm, rotated rx -180 ry 50 rz -91.34 deg; joints [-13.346, -46.758, 110.451, 133.523, 71.199, 108.744, -1078.655]
  MoveL 634 to (58.89, 251.83, 160) mm, rotated rx -180 ry 50 rz -97.9 deg; joints [-13.746, -46.768, 110.548, 133.145, 71.387, 108.806, -1072.098]
  MoveL 635 to (58.18, 244.95, 150) mm, rotated rx 180 ry 50 rz -104.5 deg; joints [-14.146, -46.776, 110.639, 132.766, 71.573, 108.868, -1065.497]
  MoveL 636 to (56.65, 238.12, 140) mm, rotated rx 180 ry 50 rz -111.11 deg; joints [-14.546, -46.781, 110.723, 132.386, 71.756, 108.933, -1058.886]
  MoveL 637 to (54.3, 231.49, 130) mm, rotated rx 180 ry 50 rz -117.7 deg; joints [-14.948, -46.784, 110.801, 132.005, 71.937, 108.999, -1052.295]
  MoveL 638 to (51.17, 225.17, 120) mm, rotated rx -180 ry 50 rz -124.24 deg; joints [-15.349, -46.786, 110.873, 131.623, 72.114, 109.067, -1045.756]
  MoveL 639 to (47.33, 219.29, 110) mm, rotated rx 180 ry 50 rz -130.7 deg; joints [-15.751, -46.788, 110.939, 131.239, 72.288, 109.139, -1039.296]
  MoveL 640 to (42.85, 213.95, 100) mm, rotated rx -180 ry 50 rz -137.06 deg; joints [-16.154, -46.79, 110.999, 130.854, 72.459, 109.214, -1032.941]
  MoveL 641 to (37.86, 209.24, 90) mm, rotated rx 180 ry 50 rz -143.28 deg; joints [-16.557, -46.793, 111.054, 130.468, 72.625, 109.292, -1026.718]
  MoveL 642 to (32.46, 205.23, 80) mm, rotated rx -180 ry 50 rz -149.35 deg; joints [-16.96, -46.796, 111.102, 130.08, 72.788, 109.375, -1020.653]
  MoveL 643 to (26.8, 201.92, 70) mm, rotated rx 180 ry 50 rz -155.23 deg; joints [-17.364, -46.8, 111.144, 129.691, 72.947, 109.461, -1014.769]
  MoveL 644 to (21, 199.35, 60) mm, rotated rx 180 ry 50 rz -160.91 deg; joints [-17.768, -46.804, 111.18, 129.3, 73.102, 109.552, -1009.094]
  MoveL 645 to (15.19, 197.47, 50) mm, rotated rx -180 ry 50 rz -166.35 deg; joints [-18.172, -46.809, 111.211, 128.908, 73.253, 109.646, -1003.653]
  MoveL 646 to (9.5, 196.25, 40) mm, rotated rx 180 ry 50 rz -171.53 deg; joints [-18.576, -46.815, 111.235, 128.515, 73.401, 109.745, -998.473]
  MoveL 647 to (4.03, 195.62, 30) mm, rotated rx 180 ry 50 rz -176.42 deg; joints [-18.981, -46.82, 111.254, 128.122, 73.547, 109.847, -993.581]
  MoveL 648 to (-1.12, 195.49, 20) mm, rotated rx 180 ry 50 rz 179.01 deg; joints [-19.385, -46.825, 111.266, 127.727, 73.689, 109.953, -989.007]
  MoveL 649 to (-5.87, 195.78, 10) mm, rotated rx 180 ry 50 rz 174.78 deg; joints [-19.79, -46.829, 111.273, 127.331, 73.829, 110.061, -984.779]
  MoveL 650 to (-10.16, 196.36, 0) mm, rotated rx 180 ry 50 rz 170.93 deg; joints [-20.194, -46.832, 111.273, 126.935, 73.966, 110.173, -980.929]
  MoveL 651 to (28.22, 306.19, 290) mm, rotated rx 180 ry 50 rz -31.42 deg; joints [-8.613, -46.241, 108.793, 138.013, 68.889, 107.96, -1138.582]
  Set speed (60.0 mm/s)
  MoveL 652 to (-21.11, 309.47, 290) mm, rotated rx -180 ry 50 rz 23.11 deg; joints [-8.613, -46.26, 108.794, 138.009, 68.876, 107.972, -1193.11]
  MoveL 653 to (-10.16, 196.36, 0) mm, rotated rx -180 ry 50 rz 170.93 deg; joints [-20.194, -46.832, 111.273, 126.935, 73.966, 110.173, -1340.929]
  Set speed (60.0 mm/s)
  MoveL 654 to (37.62, 209.05, 0) mm, rotated rx 180 ry 50 rz -143.56 deg; joints [-20.194, -46.894, 111.278, 126.922, 73.932, 110.22, -1386.442]
  MoveL 655 to (-10.16, 196.36, 0) mm, rotated rx 180 ry 50 rz 170.93 deg; joints [-20.194, -46.832, 111.273, 126.935, 73.966, 110.173, -1340.929]
  Set speed (60.0 mm/s)
  MoveL 656 to (-5.87, 195.78, 10) mm, rotated rx -180 ry 50 rz 174.78 deg; joints [-19.79, -46.829, 111.273, 127.331, 73.829, 110.061, -1344.779]
  MoveL 657 to (-1.12, 195.49, 20) mm, rotated rx -180 ry 50 rz 179.01 deg; joints [-19.385, -46.825, 111.266, 127.727, 73.689, 109.953, -1349.007]
